KUKA KRL program: EPS_2_25694_AC01A_A_20260223033028.src

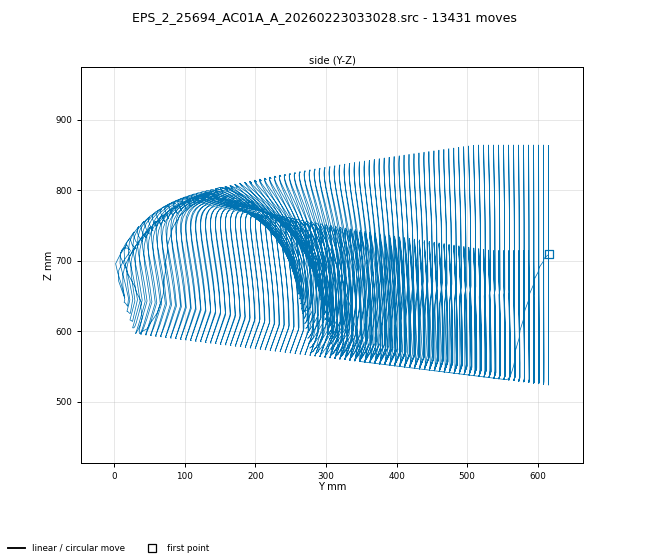
[picture p0: tool path of EPS_2_25694_AC01A_A_20260223033028.src, 13431 of 13433 moves have a stored position in this frame; points joined in program order, loops and branches not executed]
&ACCESS RVP
&REL 4
&COMMENT QRS 19112012
&PARAM EDITMASK = *
DEF PART()
EXT BAS (BAS_COMMAND :IN,REAL :IN )
INT I
BAS (#INITMOV,0 )

;KUKA QRS Post kuka4.cps  Date:22-06-2017 !

File_ID=3047

QRS_PRE_INIT()

;Init var - Until changes are made in qrs_pre_init
Outlet_Square_prg=0
Inlet_1_Square_prg=0
Inlet_2_Square_prg=0
Inlet_3_Square_prg=0
Inlet_4_Square_prg=0
Inlet_5_Square_prg=0

Outlet_1={X 0.000, Y 513.730, Z 763.500, B 0.000, E1 0.000 }
Inlet_1={X 0.000, Y 535.920, Z 314.500, B 0.000, E1 93.000 }
Inlet_2={X 0.000, Y 525.250, Z 538.500, B 0.000, E1 257.000 }
Outlet_1_type=201
Inlet_1_type=299
Inlet_2_type=251
;QRS#1=Sidecore dimensions
;QRS#2=200-8" PVC SDR 35
;QRS#3=300-12" PVC SDR 35
;QRS#4=250-10" PVC SDR 35
;QRS#5=
;QRS#6=
;QRS#7=
;QRS#8=
;QRS#9=12-08 PSX
;QRS#10=16M PSX
;QRS#11=14M PSX
;QRS#12=
;QRS#13=
;QRS#14=
;QRS#15=
;QRS#16=1220x127x1143 3,75'
;QRS#17=EPS Height
;QRS#18=864
;QRS#19=*
;QRS#20= UPDATED VERSION 22-06-2017
;QRS#21=*
Outlet_Square=0100
Inlet_1_Square=0150
Inlet_2_Square=0100
Inlet_3_Square=0
Inlet_4_Square=0
Inlet_5_Square=0
Mill_Square=1
Outlet_Square_Prg=204
Inlet_1_Square_prg=206
Inlet_2_Square_prg=205

QRS_INIT()

$ADVANCE=5

; T1
PTP {E1 173.417,E2 173.417}
PTP {X 0,Y 615.495,A -85,B 0,C 180,E1 173.417,E2 173.417,E3 0,E4 0,E5 0,E6 0}
QRS_SPEED_INIT()
LIN {X 0,Y 615.495,Z 709.245,A -85,B 0,C 180,E1 173.417,E2 173.417,E3 0,E4 0,E5 0,E6 0} C_VEL
LIN {X 0,Y 615.493,Z 705.573,A -85,B 0,C 180,E1 172.125,E2 172.125} C_VEL
LIN {X 0,Y 615.497,Z 700.547,A -85,B 0,C 180,E1 170.802,E2 170.802} C_VEL
LIN {X 0,Y 615.496,Z 694.074,A -85,B 0,C 180,E1 169.474,E2 169.474} C_VEL
LIN {X 0,Y 615.496,Z 685.953,A -85,B 0,C 180,E1 168.14,E2 168.14} C_VEL
LIN {X 0,Y 615.496,Z 677.25,A -85,B 0,C 180,E1 166.967,E2 166.967} C_VEL
LIN {X 0,Y 615.496,Z 667.933,A -85,B 0,C 180,E1 165.912,E2 165.912} C_VEL
LIN {X 0,Y 615.497,Z 657.856,A -85,B 0,C 180,E1 164.944,E2 164.944} C_VEL
LIN {X 0,Y 615.499,Z 645.706,A -85,B 0,C 180,E1 163.964,E2 163.964} C_VEL
LIN {X 0,Y 615.497,Z 633.795,A -85,B 0,C 180,E1 163.158,E2 163.158} C_VEL
LIN {X 0,Y 615.489,Z 621.694,A -85,B 0,C 180,E1 162.473,E2 162.473} C_VEL
LIN {X 0,Y 615.478,Z 607.053,A -85,B 0,C 180,E1 161.801,E2 161.801} C_VEL
LIN {X 0,Y 615.487,Z 591.984,A -85,B 0,C 180,E1 161.268,E2 161.268} C_VEL
LIN {X 0,Y 615.48,Z 576.911,A -85,B 0,C 180,E1 160.879,E2 160.879} C_VEL
LIN {X 0,Y 615.476,Z 561.369,A -85,B 0,C 180,E1 160.619,E2 160.619} C_VEL
LIN {X 0,Y 615.5,Z 523.699,A -85,B 0,C 180,E1 160.164,E2 160.164} C_VEL
LIN {X 0,Y 615.486,Z 523.681,A -85,B 0,C 180,E1 157.156,E2 157.156} C_VEL
LIN {X 0,Y 615.484,Z 523.694,A -85,B 0,C 180,E1 154.284,E2 154.284} C_VEL
LIN {X 0,Y 615.478,Z 523.69,A -85,B 0,C 180,E1 151.552,E2 151.552} C_VEL
LIN {X 0,Y 615.484,Z 523.682,A -85,B 0,C 180,E1 148.915,E2 148.915} C_VEL
LIN {X 0,Y 615.496,Z 523.697,A -85,B 0,C 180,E1 145.979,E2 145.979} C_VEL
LIN {X 0,Y 615.487,Z 523.682,A -85,B 0,C 180,E1 143.064,E2 143.064} C_VEL
LIN {X 0,Y 615.477,Z 523.69,A -85,B 0,C 180,E1 140.249,E2 140.249} C_VEL
LIN {X 0,Y 615.493,Z 523.698,A -85,B 0,C 180,E1 137.648,E2 137.648} C_VEL
LIN {X 0,Y 615.481,Z 523.684,A -85,B 0,C 180,E1 134.931,E2 134.931} C_VEL
LIN {X 0,Y 615.477,Z 523.69,A -85,B 0,C 180,E1 132.08,E2 132.08} C_VEL
LIN {X 0,Y 615.492,Z 523.695,A -85,B 0,C 180,E1 129.75,E2 129.75} C_VEL
LIN {X 0,Y 615.482,Z 523.686,A -85,B 0,C 180,E1 126.936,E2 126.936} C_VEL
LIN {X 0,Y 615.49,Z 523.681,A -85,B 0,C 180,E1 124.702,E2 124.702} C_VEL
LIN {X 0,Y 615.484,Z 523.682,A -85,B 0,C 180,E1 122.331,E2 122.331} C_VEL
LIN {X 0,Y 615.495,Z 523.701,A -85,B 0,C 180,E1 119.406,E2 119.406} C_VEL
LIN {X 0,Y 615.492,Z 523.68,A -85,B 0,C 180,E1 116.444,E2 116.444} C_VEL
LIN {X 0,Y 615.487,Z 523.693,A -85,B 0,C 180,E1 113.557,E2 113.557} C_VEL
LIN {X 0,Y 615.481,Z 523.688,A -85,B 0,C 180,E1 110.731,E2 110.731} C_VEL
LIN {X 0,Y 615.478,Z 523.684,A -85,B 0,C 180,E1 107.958,E2 107.958} C_VEL
LIN {X 0,Y 615.495,Z 523.698,A -85,B 0,C 180,E1 105.226,E2 105.226} C_VEL
LIN {X 0,Y 615.483,Z 523.686,A -85,B 0,C 180,E1 102.531,E2 102.531} C_VEL
LIN {X 0,Y 615.48,Z 523.683,A -85,B 0,C 180,E1 99.863,E2 99.863} C_VEL
LIN {X 0,Y 615.49,Z 523.694,A -85,B 0,C 180,E1 97.216,E2 97.216} C_VEL
LIN {X 0,Y 615.481,Z 523.692,A -85,B 0,C 180,E1 94.585,E2 94.585} C_VEL
LIN {X 0,Y 615.494,Z 523.68,A -85,B 0,C 180,E1 91.963,E2 91.963} C_VEL
LIN {X 0,Y 615.476,Z 523.689,A -85,B 0,C 180,E1 89.346,E2 89.346} C_VEL
LIN {X 0,Y 615.492,Z 523.699,A -85,B 0,C 180,E1 86.727,E2 86.727} C_VEL
LIN {X 0,Y 615.487,Z 523.684,A -85,B 0,C 180,E1 84.102,E2 84.102} C_VEL
LIN {X 0,Y 615.477,Z 523.685,A -85,B 0,C 180,E1 81.464,E2 81.464} C_VEL
LIN {X 0,Y 615.498,Z 523.694,A -85,B 0,C 180,E1 78.808,E2 78.808} C_VEL
LIN {X 0,Y 615.485,Z 523.686,A -85,B 0,C 180,E1 76.067,E2 76.067} C_VEL
LIN {X 0,Y 615.478,Z 523.684,A -85,B 0,C 180,E1 73.414,E2 73.414} C_VEL
LIN {X 0,Y 615.492,Z 523.696,A -85,B 0,C 180,E1 70.663,E2 70.663} C_VEL
LIN {X 0,Y 615.491,Z 523.681,A -85,B 0,C 180,E1 67.652,E2 67.652} C_VEL
LIN {X 0,Y 615.475,Z 523.687,A -85,B 0,C 180,E1 65.008,E2 65.008} C_VEL
LIN {X 0,Y 615.481,Z 523.689,A -85,B 0,C 180,E1 62.823,E2 62.823} C_VEL
LIN {X 0,Y 615.492,Z 523.698,A -85,B 0,C 180,E1 60.204,E2 60.204} C_VEL
LIN {X 0,Y 615.491,Z 523.682,A -85,B 0,C 180,E1 57.543,E2 57.543} C_VEL
LIN {X 0,Y 615.482,Z 523.682,A -85,B 0,C 180,E1 55.185,E2 55.185} C_VEL
LIN {X 0,Y 615.475,Z 523.688,A -85,B 0,C 180,E1 52.758,E2 52.758} C_VEL
LIN {X 0,Y 615.488,Z 523.695,A -85,B 0,C 180,E1 49.91,E2 49.91} C_VEL
LIN {X 0,Y 615.485,Z 523.689,A -85,B 0,C 180,E1 47.647,E2 47.647} C_VEL
LIN {X 0,Y 615.478,Z 523.683,A -85,B 0,C 180,E1 44.931,E2 44.931} C_VEL
LIN {X 0,Y 615.498,Z 523.696,A -85,B 0,C 180,E1 42.082,E2 42.082} C_VEL
LIN {X 0,Y 615.492,Z 523.68,A -85,B 0,C 180,E1 39.063,E2 39.063} C_VEL
LIN {X 0,Y 615.479,Z 523.687,A -85,B 0,C 180,E1 36.425,E2 36.425} C_VEL
LIN {X 0,Y 615.487,Z 523.692,A -85,B 0,C 180,E1 33.535,E2 33.535} C_VEL
LIN {X 0,Y 615.485,Z 523.682,A -85,B 0,C 180,E1 30.919,E2 30.919} C_VEL
LIN {X 0,Y 615.476,Z 523.685,A -85,B 0,C 180,E1 28.449,E2 28.449} C_VEL
LIN {X 0,Y 615.496,Z 523.701,A -85,B 0,C 180,E1 27.706,E2 27.706} C_VEL
LIN {X 0,Y 615.489,Z 531.805,A -85,B 0,C 180,E1 27.591,E2 27.591} C_VEL
LIN {X 0,Y 615.495,Z 589.214,A -85,B 0,C 180,E1 26.895,E2 26.895} C_VEL
LIN {X 0,Y 615.478,Z 603.233,A -85,B 0,C 180,E1 26.595,E2 26.595} C_VEL
LIN {X 0,Y 615.483,Z 616.816,A -85,B 0,C 180,E1 26.17,E2 26.17} C_VEL
LIN {X 0,Y 615.496,Z 629.536,A -85,B 0,C 180,E1 25.643,E2 25.643} C_VEL
LIN {X 0,Y 615.491,Z 641.959,A -85,B 0,C 180,E1 24.991,E2 24.991} C_VEL
LIN {X 0,Y 615.498,Z 653.128,A -85,B 0,C 180,E1 24.271,E2 24.271} C_VEL
LIN {X 0,Y 615.499,Z 664.53,A -85,B 0,C 180,E1 23.377,E2 23.377} C_VEL
LIN {X 0,Y 615.492,Z 675.308,A -85,B 0,C 180,E1 22.348,E2 22.348} C_VEL
LIN {X 0,Y 615.496,Z 684.638,A -85,B 0,C 180,E1 21.256,E2 21.256} C_VEL
LIN {X 0,Y 615.494,Z 691.433,A -85,B 0,C 180,E1 20.296,E2 20.296} C_VEL
LIN {X 0,Y 615.495,Z 697.081,A -85,B 0,C 180,E1 19.337,E2 19.337} C_VEL
LIN {X 0,Y 615.495,Z 702.21,A -85,B 0,C 180,E1 18.282,E2 18.282} C_VEL
LIN {X 0,Y 615.496,Z 707.259,A -85,B 0,C 180,E1 16.928,E2 16.928} C_VEL
LIN {X 0,Y 615.494,Z 710.032,A -85,B 0,C 180,E1 15.905,E2 15.905} C_VEL
LIN {X 0,Y 615.496,Z 712.389,A -85,B 0,C 180,E1 14.549,E2 14.549} C_VEL
LIN {X 0,Y 615.489,Z 713.337,A -85,B 0,C 180,E1 13.201,E2 13.201} C_VEL
LIN {X 0,Y 615.495,Z 712.911,A -85,B 0,C 180,E1 11.86,E2 11.86} C_VEL
LIN {X 0,Y 615.496,Z 711.131,A -85,B 0,C 180,E1 10.526,E2 10.526} C_VEL
LIN {X 0,Y 615.496,Z 707.948,A -85,B 0,C 180,E1 9.198,E2 9.198} C_VEL
LIN {X 0,Y 615.493,Z 703.274,A -85,B 0,C 180,E1 7.875,E2 7.875} C_VEL
LIN {X 0,Y 615.497,Z 696.991,A -85,B 0,C 180,E1 6.556,E2 6.556} C_VEL
LIN {X 0,Y 615.495,Z 690.024,A -85,B 0,C 180,E1 5.405,E2 5.405} C_VEL
LIN {X 0,Y 615.497,Z 681.428,A -85,B 0,C 180,E1 4.256,E2 4.256} C_VEL
LIN {X 0,Y 615.496,Z 672.486,A -85,B 0,C 180,E1 3.273,E2 3.273} C_VEL
LIN {X 0,Y 615.499,Z 661.696,A -85,B 0,C 180,E1 2.29,E2 2.29} C_VEL
LIN {X 0,Y 615.498,Z 650.756,A -85,B 0,C 180,E1 1.472,E2 1.472} C_VEL
LIN {X 0,Y 615.488,Z 638.756,A -85,B 0,C 180,E1 0.736,E2 0.736} C_VEL
LIN {X 0,Y 615.485,Z 625.402,A -85,B 0,C 180,E1 0.081,E2 0.081} C_VEL
LIN {X 0,Y 615.495,Z 611.227,A -85,B 0,C 180,E1 -0.45,E2 -0.45} C_VEL
LIN {X 0,Y 615.48,Z 597.695,A -85,B 0,C 180,E1 -0.818,E2 -0.818} C_VEL
LIN {X 0,Y 615.476,Z 583.862,A -85,B 0,C 180,E1 -1.064,E2 -1.064} C_VEL
LIN {X 0,Y 615.488,Z 523.701,A -85,B 0,C 180,E1 -1.779,E2 -1.779} C_VEL
LIN {X 0,Y 615.497,Z 523.68,A -85,B 0,C 180,E1 -4.585,E2 -4.585} C_VEL
LIN {X 0,Y 615.477,Z 523.691,A -85,B 0,C 180,E1 -7.216,E2 -7.216} C_VEL
LIN {X 0,Y 615.485,Z 523.695,A -85,B 0,C 180,E1 -9.863,E2 -9.863} C_VEL
LIN {X 0,Y 615.486,Z 523.683,A -85,B 0,C 180,E1 -12.53,E2 -12.53} C_VEL
LIN {X 0,Y 615.478,Z 523.694,A -85,B 0,C 180,E1 -15.227,E2 -15.227} C_VEL
LIN {X 0,Y 615.487,Z 523.689,A -85,B 0,C 180,E1 -17.957,E2 -17.957} C_VEL
LIN {X 0,Y 615.49,Z 523.683,A -85,B 0,C 180,E1 -20.731,E2 -20.731} C_VEL
LIN {X 0,Y 615.489,Z 523.699,A -85,B 0,C 180,E1 -23.557,E2 -23.557} C_VEL
LIN {X 0,Y 615.494,Z 523.691,A -85,B 0,C 180,E1 -25.716,E2 -25.716} C_VEL
LIN {X 0,Y 615.476,Z 523.685,A -85,B 0,C 180,E1 -28.449,E2 -28.449} C_VEL
LIN {X 0,Y 615.491,Z 523.692,A -85,B 0,C 180,E1 -31.088,E2 -31.088} C_VEL
LIN {X 0,Y 615.497,Z 523.682,A -85,B 0,C 180,E1 -34.022,E2 -34.022} C_VEL
LIN {X 0,Y 615.482,Z 523.692,A -85,B 0,C 180,E1 -36.937,E2 -36.937} C_VEL
LIN {X 0,Y 615.481,Z 523.689,A -85,B 0,C 180,E1 -39.751,E2 -39.751} C_VEL
LIN {X 0,Y 615.488,Z 523.682,A -85,B 0,C 180,E1 -42.353,E2 -42.353} C_VEL
LIN {X 0,Y 615.488,Z 523.698,A -85,B 0,C 180,E1 -45.069,E2 -45.069} C_VEL
LIN {X 0,Y 615.477,Z 523.686,A -85,B 0,C 180,E1 -47.921,E2 -47.921} C_VEL
LIN {X 0,Y 615.493,Z 523.681,A -85,B 0,C 180,E1 -50.251,E2 -50.251} C_VEL
LIN {X 0,Y 615.492,Z 523.701,A -85,B 0,C 180,E1 -53.063,E2 -53.063} C_VEL
LIN {X 0,Y 615.497,Z 523.692,A -85,B 0,C 180,E1 -55.299,E2 -55.299} C_VEL
LIN {X 0,Y 615.484,Z 523.686,A -85,B 0,C 180,E1 -57.67,E2 -57.67} C_VEL
LIN {X 0,Y 615.483,Z 523.872,A -85,B 0,C 180,E1 -60.304,E2 -60.304} C_VEL
LIN {X 0,Y 615.491,Z 544.028,A -85,B 0,C 180,E1 -63.106,E2 -63.106} C_VEL
LIN {X 0,Y 615.489,Z 563.357,A -85,B 0,C 180,E1 -65.729,E2 -65.729} C_VEL
LIN {X 0,Y 615.494,Z 584.743,A -85,B 0,C 180,E1 -68.569,E2 -68.569} C_VEL
LIN {X 0,Y 615.488,Z 606.431,A -85,B 0,C 180,E1 -71.396,E2 -71.396} C_VEL
LIN {X 0,Y 615.479,Z 627.455,A -85,B 0,C 180,E1 -74.095,E2 -74.095} C_VEL
LIN {X 0,Y 615.492,Z 650.105,A -85,B 0,C 180,E1 -76.967,E2 -76.967} C_VEL
LIN {X 0,Y 615.488,Z 651.269,A -85,B 0,C 180,E1 -77.114,E2 -77.114} C_VEL
LIN {X 0,Y 615.489,Z 759.854,A -85,B 0,C 180,E1 -78.411,E2 -78.411} C_VEL
LIN {X 0,Y 615.492,Z 772.359,A -85,B 0,C 180,E1 -78.682,E2 -78.682} C_VEL
LIN {X 0,Y 615.496,Z 785.512,A -85,B 0,C 180,E1 -79.109,E2 -79.109} C_VEL
LIN {X 0,Y 615.484,Z 797.486,A -85,B 0,C 180,E1 -79.64,E2 -79.64} C_VEL
LIN {X 0,Y 615.483,Z 809.002,A -85,B 0,C 180,E1 -80.304,E2 -80.304} C_VEL
LIN {X 0,Y 615.499,Z 819.346,A -85,B 0,C 180,E1 -81.05,E2 -81.05} C_VEL
LIN {X 0,Y 615.497,Z 827.816,A -85,B 0,C 180,E1 -81.795,E2 -81.795} C_VEL
LIN {X 0,Y 615.498,Z 835.61,A -85,B 0,C 180,E1 -82.62,E2 -82.62} C_VEL
LIN {X 0,Y 615.496,Z 843.206,A -85,B 0,C 180,E1 -83.608,E2 -83.608} C_VEL
LIN {X 0,Y 615.498,Z 850.207,A -85,B 0,C 180,E1 -84.759,E2 -84.759} C_VEL
LIN {X 0,Y 615.494,Z 854.853,A -85,B 0,C 180,E1 -85.744,E2 -85.744} C_VEL
LIN {X 0,Y 615.496,Z 858.4,A -85,B 0,C 180,E1 -86.727,E2 -86.727} C_VEL
LIN {X 0,Y 615.497,Z 860.234,A -85,B 0,C 180,E1 -87.383,E2 -87.383} C_VEL
LIN {X 0,Y 615.496,Z 861.609,A -85,B 0,C 180,E1 -88.037,E2 -88.037} C_VEL
LIN {X 0,Y 615.496,Z 863.174,A -85,B 0,C 180,E1 -89.346,E2 -89.346} C_VEL
LIN {X 0,Y 615.494,Z 863.389,A -85,B 0,C 180,E1 -90,E2 -90} C_VEL
LIN {X 0,Y 615.496,Z 862.579,A -85,B 0,C 180,E1 -91.309,E2 -91.309} C_VEL
LIN {X 0,Y 615.496,Z 861.608,A -85,B 0,C 180,E1 -91.963,E2 -91.963} C_VEL
LIN {X 0,Y 615.497,Z 860.232,A -85,B 0,C 180,E1 -92.618,E2 -92.618} C_VEL
LIN {X 0,Y 615.496,Z 857.348,A -85,B 0,C 180,E1 -93.601,E2 -93.601} C_VEL
LIN {X 0,Y 615.498,Z 853.44,A -85,B 0,C 180,E1 -94.585,E2 -94.585} C_VEL
LIN {X 0,Y 615.499,Z 848.403,A -85,B 0,C 180,E1 -95.57,E2 -95.57} C_VEL
LIN {X 0,Y 615.497,Z 841.87,A -85,B 0,C 180,E1 -96.583,E2 -96.583} C_VEL
LIN {X 0,Y 615.497,Z 834.13,A -85,B 0,C 180,E1 -97.546,E2 -97.546} C_VEL
LIN {X 0,Y 615.498,Z 826.041,A -85,B 0,C 180,E1 -98.371,E2 -98.371} C_VEL
LIN {X 0,Y 615.499,Z 816.163,A -85,B 0,C 180,E1 -99.199,E2 -99.199} C_VEL
LIN {X 0,Y 615.486,Z 804.975,A -85,B 0,C 180,E1 -99.946,E2 -99.946} C_VEL
LIN {X 0,Y 615.483,Z 794.015,A -85,B 0,C 180,E1 -100.527,E2 -100.527} C_VEL
LIN {X 0,Y 615.496,Z 781.426,A -85,B 0,C 180,E1 -101.042,E2 -101.042} C_VEL
LIN {X 0,Y 615.49,Z 769.049,A -85,B 0,C 180,E1 -101.402,E2 -101.402} C_VEL
LIN {X 0,Y 615.49,Z 755.439,A -85,B 0,C 180,E1 -101.652,E2 -101.652} C_VEL
LIN {X 0,Y 615.488,Z 651.263,A -85,B 0,C 180,E1 -102.887,E2 -102.887} C_VEL
LIN {X 0,Y 615.482,Z 630.116,A -85,B 0,C 180,E1 -105.566,E2 -105.566} C_VEL
LIN {X 0,Y 615.498,Z 608.936,A -85,B 0,C 180,E1 -108.28,E2 -108.28} C_VEL
LIN {X 0,Y 615.497,Z 587.409,A -85,B 0,C 180,E1 -111.081,E2 -111.081} C_VEL
LIN {X 0,Y 615.476,Z 567.021,A -85,B 0,C 180,E1 -113.781,E2 -113.781} C_VEL
LIN {X 0,Y 615.496,Z 546.216,A -85,B 0,C 180,E1 -116.594,E2 -116.594} C_VEL
LIN {X 0,Y 615.497,Z 525.925,A -85,B 0,C 180,E1 -119.406,E2 -119.406} C_VEL
LIN {X 0,Y 615.479,Z 523.686,A -85,B 0,C 180,E1 -119.744,E2 -119.744} C_VEL
LIN {X 0,Y 615.487,Z 523.688,A -85,B 0,C 180,E1 -122.458,E2 -122.458} C_VEL
LIN {X 0,Y 615.497,Z 523.696,A -85,B 0,C 180,E1 -124.815,E2 -124.815} C_VEL
LIN {X 0,Y 615.486,Z 523.691,A -85,B 0,C 180,E1 -127.243,E2 -127.243} C_VEL
LIN {X 0,Y 615.477,Z 523.686,A -85,B 0,C 180,E1 -130.087,E2 -130.087} C_VEL
LIN {X 0,Y 615.478,Z 523.691,A -85,B 0,C 180,E1 -132.354,E2 -132.354} C_VEL
LIN {X 0,Y 615.481,Z 523.694,A -85,B 0,C 180,E1 -135.069,E2 -135.069} C_VEL
LIN {X 0,Y 615.491,Z 523.682,A -85,B 0,C 180,E1 -137.92,E2 -137.92} C_VEL
LIN {X 0,Y 615.492,Z 523.693,A -85,B 0,C 180,E1 -140.938,E2 -140.938} C_VEL
LIN {X 0,Y 615.478,Z 523.685,A -85,B 0,C 180,E1 -143.574,E2 -143.574} C_VEL
LIN {X 0,Y 615.489,Z 523.697,A -85,B 0,C 180,E1 -146.466,E2 -146.466} C_VEL
LIN {X 0,Y 615.487,Z 523.687,A -85,B 0,C 180,E1 -149.08,E2 -149.08} C_VEL
LIN {X 0,Y 615.476,Z 523.685,A -85,B 0,C 180,E1 -151.552,E2 -151.552} C_VEL
LIN {X 0,Y 615.498,Z 523.699,A -85,B 0,C 180,E1 -154.43,E2 -154.43} C_VEL
LIN {X 0,Y 615.486,Z 523.684,A -85,B 0,C 180,E1 -157.155,E2 -157.155} C_VEL
LIN {X 0,Y 615.485,Z 523.69,A -85,B 0,C 180,E1 -159.967,E2 -159.967} C_VEL
LIN {X 0,Y 615.48,Z 523.692,A -85,B 0,C 180,E1 -162.729,E2 -162.729} C_VEL
LIN {X 0,Y 615.48,Z 523.684,A -85,B 0,C 180,E1 -165.45,E2 -165.45} C_VEL
LIN {X 0,Y 615.487,Z 523.701,A -85,B 0,C 180,E1 -166.252,E2 -166.252} C_VEL
LIN {X 0,Y 615.476,Z 569.038,A -85,B 0,C 180,E1 -166.819,E2 -166.819} C_VEL
LIN {X 0,Y 615.485,Z 583.996,A -85,B 0,C 180,E1 -167.134,E2 -167.134} C_VEL
LIN {X 0,Y 615.479,Z 599.217,A -85,B 0,C 180,E1 -167.595,E2 -167.595} C_VEL
LIN {X 0,Y 615.486,Z 612.817,A -85,B 0,C 180,E1 -168.139,E2 -168.139} C_VEL
LIN {X 0,Y 615.493,Z 626.215,A -85,B 0,C 180,E1 -168.807,E2 -168.807} C_VEL
LIN {X 0,Y 615.5,Z 638.582,A -85,B 0,C 180,E1 -169.556,E2 -169.556} C_VEL
LIN {X 0,Y 615.499,Z 651.123,A -85,B 0,C 180,E1 -170.47,E2 -170.47} C_VEL
LIN {X 0,Y 615.496,Z 662.521,A -85,B 0,C 180,E1 -171.463,E2 -171.463} C_VEL
LIN {X 0,Y 615.495,Z 672.115,A -85,B 0,C 180,E1 -172.454,E2 -172.454} C_VEL
LIN {X 0,Y 615.494,Z 681.536,A -85,B 0,C 180,E1 -173.608,E2 -173.608} C_VEL
LIN {X 0,Y 615.494,Z 690.39,A -85,B 0,C 180,E1 -174.923,E2 -174.923} C_VEL
LIN {X 0,Y 615.492,Z 696.739,A -85,B 0,C 180,E1 -176.071,E2 -176.071} C_VEL
LIN {X 0,Y 615.496,Z 702.589,A -85,B 0,C 180,E1 -177.382,E2 -177.382} C_VEL
LIN {X 0,Y 615.496,Z 707.094,A -85,B 0,C 180,E1 -178.691,E2 -178.691} C_VEL
LIN {X 0,Y 615.49,Z 710.314,A -85,B 0,C 180,E1 -180,E2 -180} C_VEL
LIN {X 0,Y 615.491,Z 712.362,A -85,B 0,C 180,E1 -181.308,E2 -181.308} C_VEL
LIN {X 0,Y 615.497,Z 713.291,A -85,B 0,C 180,E1 -182.618,E2 -182.618} C_VEL
LIN {X 0,Y 615.488,Z 713.108,A -85,B 0,C 180,E1 -183.928,E2 -183.928} C_VEL
LIN {X 0,Y 615.489,Z 711.806,A -85,B 0,C 180,E1 -185.241,E2 -185.241} C_VEL
LIN {X 0,Y 615.495,Z 709.245,A -85,B 0,C 180,E1 -186.583,E2 -186.583} C_VEL
LIN {X 0,Y 614.809,Z 708.026,A -85,B 0,C 180,E1 -187.114,E2 -187.114} C_VEL
LIN {X 0,Y 611.951,Z 705.822,A -85,B 0,C 180,E1 -187.974,E2 -187.974} C_VEL
LIN {X 0,Y 609.544,Z 703.512,A -85,B 0,C 180,E1 -188.657,E2 -188.657} C_VEL
LIN {X 0,Y 608.513,Z 701.422,A -85,B 0,C 180,E1 -189.174,E2 -189.174} C_VEL
LIN {X 0,Y 608.428,Z 700.673,A -85,B 0,C 180,E1 -189.347,E2 -189.347} C_VEL
LIN {X 0,Y 608.436,Z 694.266,A -85,B 0,C 180,E1 -190.65,E2 -190.65} C_VEL
LIN {X 0,Y 608.462,Z 687.154,A -85,B 0,C 180,E1 -191.83,E2 -191.83} C_VEL
LIN {X 0,Y 608.465,Z 678.57,A -85,B 0,C 180,E1 -193.016,E2 -193.016} C_VEL
LIN {X 0,Y 608.485,Z 668.197,A -85,B 0,C 180,E1 -194.207,E2 -194.207} C_VEL
LIN {X 0,Y 608.495,Z 657.544,A -85,B 0,C 180,E1 -195.233,E2 -195.233} C_VEL
LIN {X 0,Y 608.537,Z 645.262,A -85,B 0,C 180,E1 -196.225,E2 -196.225} C_VEL
LIN {X 0,Y 608.555,Z 631.774,A -85,B 0,C 180,E1 -197.127,E2 -197.127} C_VEL
LIN {X 0,Y 608.578,Z 617.426,A -85,B 0,C 180,E1 -197.907,E2 -197.907} C_VEL
LIN {X 0,Y 608.615,Z 603.979,A -85,B 0,C 180,E1 -198.493,E2 -198.493} C_VEL
LIN {X 0,Y 608.657,Z 589.173,A -85,B 0,C 180,E1 -198.994,E2 -198.994} C_VEL
LIN {X 0,Y 608.663,Z 573.906,A -85,B 0,C 180,E1 -199.366,E2 -199.366} C_VEL
LIN {X 0,Y 608.67,Z 556.486,A -85,B 0,C 180,E1 -199.629,E2 -199.629} C_VEL
LIN {X 0,Y 608.53,Z 525.02,A -85,B 0,C 180,E1 -200.013,E2 -200.013} C_VEL
LIN {X 0,Y 608.469,Z 524.693,A -85,B 0,C 180,E1 -200.053,E2 -200.053} C_VEL
LIN {X 0,Y 608.461,Z 524.688,A -85,B 0,C 180,E1 -202.476,E2 -202.476} C_VEL
LIN {X 0,Y 608.452,Z 524.688,A -85,B 0,C 180,E1 -204.571,E2 -204.571} C_VEL
LIN {X 0,Y 608.476,Z 524.684,A -85,B 0,C 180,E1 -207.206,E2 -207.206} C_VEL
LIN {X 0,Y 608.468,Z 524.695,A -85,B 0,C 180,E1 -209.971,E2 -209.971} C_VEL
LIN {X 0,Y 608.453,Z 524.687,A -85,B 0,C 180,E1 -212.879,E2 -212.879} C_VEL
LIN {X 0,Y 608.434,Z 524.689,A -85,B 0,C 180,E1 -215.278,E2 -215.278} C_VEL
LIN {X 0,Y 608.472,Z 524.688,A -85,B 0,C 180,E1 -217.746,E2 -217.746} C_VEL
LIN {X 0,Y 608.453,Z 524.696,A -85,B 0,C 180,E1 -220.329,E2 -220.329} C_VEL
LIN {X 0,Y 608.484,Z 524.683,A -85,B 0,C 180,E1 -223.31,E2 -223.31} C_VEL
LIN {X 0,Y 608.465,Z 524.693,A -85,B 0,C 180,E1 -226.13,E2 -226.13} C_VEL
LIN {X 0,Y 608.451,Z 524.691,A -85,B 0,C 180,E1 -228.823,E2 -228.823} C_VEL
LIN {X 0,Y 608.464,Z 524.685,A -85,B 0,C 180,E1 -231.411,E2 -231.411} C_VEL
LIN {X 0,Y 608.445,Z 524.69,A -85,B 0,C 180,E1 -233.954,E2 -233.954} C_VEL
LIN {X 0,Y 608.467,Z 524.692,A -85,B 0,C 180,E1 -236.329,E2 -236.329} C_VEL
LIN {X 0,Y 608.46,Z 524.694,A -85,B 0,C 180,E1 -238.73,E2 -238.73} C_VEL
LIN {X 0,Y 608.474,Z 524.685,A -85,B 0,C 180,E1 -241.379,E2 -241.379} C_VEL
LIN {X 0,Y 608.443,Z 524.689,A -85,B 0,C 180,E1 -243.964,E2 -243.964} C_VEL
LIN {X 0,Y 608.461,Z 524.688,A -85,B 0,C 180,E1 -246.155,E2 -246.155} C_VEL
LIN {X 0,Y 608.471,Z 524.688,A -85,B 0,C 180,E1 -248.308,E2 -248.308} C_VEL
LIN {X 0,Y 608.467,Z 524.688,A -85,B 0,C 180,E1 -251.284,E2 -251.284} C_VEL
LIN {X 0,Y 608.456,Z 524.686,A -85,B 0,C 180,E1 -253.906,E2 -253.906} C_VEL
LIN {X 0,Y 608.47,Z 524.691,A -85,B 0,C 180,E1 -256.643,E2 -256.643} C_VEL
LIN {X 0,Y 608.461,Z 524.69,A -85,B 0,C 180,E1 -259.35,E2 -259.35} C_VEL
LIN {X 0,Y 608.474,Z 524.684,A -85,B 0,C 180,E1 -262.033,E2 -262.033} C_VEL
LIN {X 0,Y 608.465,Z 524.69,A -85,B 0,C 180,E1 -264.698,E2 -264.698} C_VEL
LIN {X 0,Y 608.475,Z 524.69,A -85,B 0,C 180,E1 -267.352,E2 -267.352} C_VEL
LIN {X 0,Y 608.477,Z 524.684,A -85,B 0,C 180,E1 -270,E2 -270} C_VEL
LIN {X 0,Y 608.469,Z 524.687,A -85,B 0,C 180,E1 -272.648,E2 -272.648} C_VEL
LIN {X 0,Y 608.473,Z 524.695,A -85,B 0,C 180,E1 -275.301,E2 -275.301} C_VEL
LIN {X 0,Y 608.476,Z 524.685,A -85,B 0,C 180,E1 -277.967,E2 -277.967} C_VEL
LIN {X 0,Y 608.456,Z 524.687,A -85,B 0,C 180,E1 -280.65,E2 -280.65} C_VEL
LIN {X 0,Y 608.471,Z 524.695,A -85,B 0,C 180,E1 -283.356,E2 -283.356} C_VEL
LIN {X 0,Y 608.458,Z 524.687,A -85,B 0,C 180,E1 -286.093,E2 -286.093} C_VEL
LIN {X 0,Y 608.452,Z 524.688,A -85,B 0,C 180,E1 -288.869,E2 -288.869} C_VEL
LIN {X 0,Y 608.474,Z 524.693,A -85,B 0,C 180,E1 -291.691,E2 -291.691} C_VEL
LIN {X 0,Y 608.451,Z 524.687,A -85,B 0,C 180,E1 -294.571,E2 -294.571} C_VEL
LIN {X 0,Y 608.474,Z 524.688,A -85,B 0,C 180,E1 -297.207,E2 -297.207} C_VEL
LIN {X 0,Y 608.47,Z 524.691,A -85,B 0,C 180,E1 -299.973,E2 -299.973} C_VEL
LIN {X 0,Y 608.464,Z 524.686,A -85,B 0,C 180,E1 -302.523,E2 -302.523} C_VEL
LIN {X 0,Y 608.448,Z 524.69,A -85,B 0,C 180,E1 -305.277,E2 -305.277} C_VEL
LIN {X 0,Y 608.465,Z 524.689,A -85,B 0,C 180,E1 -308.241,E2 -308.241} C_VEL
LIN {X 0,Y 608.477,Z 524.687,A -85,B 0,C 180,E1 -310.332,E2 -310.332} C_VEL
LIN {X 0,Y 608.463,Z 524.687,A -85,B 0,C 180,E1 -313.309,E2 -313.309} C_VEL
LIN {X 0,Y 608.475,Z 524.693,A -85,B 0,C 180,E1 -316.132,E2 -316.132} C_VEL
LIN {X 0,Y 608.455,Z 524.687,A -85,B 0,C 180,E1 -318.824,E2 -318.824} C_VEL
LIN {X 0,Y 608.468,Z 524.686,A -85,B 0,C 180,E1 -321.412,E2 -321.412} C_VEL
LIN {X 0,Y 608.475,Z 524.692,A -85,B 0,C 180,E1 -323.95,E2 -323.95} C_VEL
LIN {X 0,Y 608.467,Z 524.693,A -85,B 0,C 180,E1 -326.33,E2 -326.33} C_VEL
LIN {X 0,Y 608.474,Z 524.687,A -85,B 0,C 180,E1 -328.727,E2 -328.727} C_VEL
LIN {X 0,Y 608.465,Z 524.685,A -85,B 0,C 180,E1 -331.38,E2 -331.38} C_VEL
LIN {X 0,Y 608.466,Z 524.694,A -85,B 0,C 180,E1 -332.145,E2 -332.145} C_VEL
LIN {X 0,Y 608.622,Z 556.104,A -85,B 0,C 180,E1 -332.53,E2 -332.53} C_VEL
LIN {X 0,Y 608.627,Z 589.449,A -85,B 0,C 180,E1 -332.948,E2 -332.948} C_VEL
LIN {X 0,Y 608.578,Z 603.495,A -85,B 0,C 180,E1 -333.255,E2 -333.255} C_VEL
LIN {X 0,Y 608.564,Z 616.069,A -85,B 0,C 180,E1 -333.648,E2 -333.648} C_VEL
LIN {X 0,Y 608.551,Z 629.667,A -85,B 0,C 180,E1 -334.214,E2 -334.214} C_VEL
LIN {X 0,Y 608.538,Z 642.325,A -85,B 0,C 180,E1 -334.886,E2 -334.886} C_VEL
LIN {X 0,Y 608.502,Z 654.708,A -85,B 0,C 180,E1 -335.703,E2 -335.703} C_VEL
LIN {X 0,Y 608.484,Z 665.932,A -85,B 0,C 180,E1 -336.608,E2 -336.608} C_VEL
LIN {X 0,Y 608.471,Z 676.055,A -85,B 0,C 180,E1 -337.595,E2 -337.595} C_VEL
LIN {X 0,Y 608.46,Z 685.081,A -85,B 0,C 180,E1 -338.664,E2 -338.664} C_VEL
LIN {X 0,Y 608.441,Z 692.491,A -85,B 0,C 180,E1 -339.725,E2 -339.725} C_VEL
LIN {X 0,Y 608.437,Z 698.556,A -85,B 0,C 180,E1 -340.78,E2 -340.78} C_VEL
LIN {X 0,Y 608.428,Z 703.431,A -85,B 0,C 180,E1 -341.828,E2 -341.828} C_VEL
LIN {X 0,Y 608.424,Z 707.298,A -85,B 0,C 180,E1 -342.87,E2 -342.87} C_VEL
LIN {X 0,Y 608.43,Z 710.263,A -85,B 0,C 180,E1 -343.906,E2 -343.906} C_VEL
LIN {X 0,Y 608.42,Z 712.809,A -85,B 0,C 180,E1 -345.278,E2 -345.278} C_VEL
LIN {X 0,Y 608.433,Z 713.912,A -85,B 0,C 180,E1 -346.643,E2 -346.643} C_VEL
LIN {X 0,Y 608.439,Z 713.626,A -85,B 0,C 180,E1 -348,E2 -348} C_VEL
LIN {X 0,Y 608.436,Z 711.969,A -85,B 0,C 180,E1 -349.35,E2 -349.35} C_VEL
LIN {X 0,Y 608.421,Z 708.912,A -85,B 0,C 180,E1 -350.694,E2 -350.694} C_VEL
LIN {X 0,Y 608.428,Z 704.394,A -85,B 0,C 180,E1 -352.033,E2 -352.033} C_VEL
LIN {X 0,Y 608.438,Z 699.92,A -85,B 0,C 180,E1 -353.034,E2 -353.034} C_VEL
LIN {X 0,Y 608.457,Z 693.492,A -85,B 0,C 180,E1 -354.2,E2 -354.2} C_VEL
LIN {X 0,Y 608.465,Z 685.548,A -85,B 0,C 180,E1 -355.363,E2 -355.363} C_VEL
LIN {X 0,Y 608.478,Z 677.282,A -85,B 0,C 180,E1 -356.358,E2 -356.358} C_VEL
LIN {X 0,Y 608.489,Z 667.392,A -85,B 0,C 180,E1 -357.352,E2 -357.352} C_VEL
LIN {X 0,Y 608.497,Z 656.422,A -85,B 0,C 180,E1 -358.263,E2 -358.263} C_VEL
LIN {X 0,Y 608.534,Z 644.213,A -85,B 0,C 180,E1 -359.09,E2 -359.09} C_VEL
LIN {X 0,Y 608.547,Z 632.216,A -85,B 0,C 180,E1 -359.752,E2 -359.752} C_VEL
LIN {X 0,Y 608.571,Z 619.003,A -85,B 0,C 180,E1 -360.331,E2 -360.331} C_VEL
LIN {X 0,Y 608.592,Z 604.509,A -85,B 0,C 180,E1 -360.807,E2 -360.807} C_VEL
LIN {X 0,Y 608.597,Z 590.813,A -85,B 0,C 180,E1 -361.117,E2 -361.117} C_VEL
LIN {X 0,Y 608.617,Z 565.495,A -85,B 0,C 180,E1 -361.448,E2 -361.448} C_VEL
LIN {X 0,Y 608.503,Z 525.017,A -85,B 0,C 180,E1 -361.934,E2 -361.934} C_VEL
LIN {X 0,Y 608.452,Z 524.695,A -85,B 0,C 180,E1 -361.945,E2 -361.945} C_VEL
LIN {X 0,Y 608.465,Z 524.686,A -85,B 0,C 180,E1 -364.638,E2 -364.638} C_VEL
LIN {X 0,Y 608.457,Z 524.691,A -85,B 0,C 180,E1 -367.3,E2 -367.3} C_VEL
LIN {X 0,Y 608.455,Z 524.692,A -85,B 0,C 180,E1 -369.978,E2 -369.978} C_VEL
LIN {X 0,Y 608.473,Z 524.685,A -85,B 0,C 180,E1 -372.677,E2 -372.677} C_VEL
LIN {X 0,Y 608.465,Z 524.694,A -85,B 0,C 180,E1 -375.406,E2 -375.406} C_VEL
LIN {X 0,Y 608.449,Z 524.689,A -85,B 0,C 180,E1 -378.172,E2 -378.172} C_VEL
LIN {X 0,Y 608.46,Z 524.689,A -85,B 0,C 180,E1 -380.982,E2 -380.982} C_VEL
LIN {X 0,Y 608.468,Z 524.69,A -85,B 0,C 180,E1 -383.845,E2 -383.845} C_VEL
LIN {X 0,Y 608.446,Z 524.69,A -85,B 0,C 180,E1 -386.036,E2 -386.036} C_VEL
LIN {X 0,Y 608.466,Z 524.686,A -85,B 0,C 180,E1 -388.62,E2 -388.62} C_VEL
LIN {X 0,Y 608.477,Z 524.694,A -85,B 0,C 180,E1 -391.316,E2 -391.316} C_VEL
LIN {X 0,Y 608.478,Z 524.688,A -85,B 0,C 180,E1 -393.737,E2 -393.737} C_VEL
LIN {X 0,Y 608.457,Z 524.687,A -85,B 0,C 180,E1 -396.092,E2 -396.092} C_VEL
LIN {X 0,Y 608.469,Z 524.686,A -85,B 0,C 180,E1 -398.588,E2 -398.588} C_VEL
LIN {X 0,Y 608.46,Z 524.695,A -85,B 0,C 180,E1 -401.343,E2 -401.343} C_VEL
LIN {X 0,Y 608.46,Z 524.686,A -85,B 0,C 180,E1 -404.265,E2 -404.265} C_VEL
LIN {X 0,Y 608.45,Z 524.696,A -85,B 0,C 180,E1 -407.041,E2 -407.041} C_VEL
LIN {X 0,Y 608.451,Z 524.69,A -85,B 0,C 180,E1 -409.697,E2 -409.697} C_VEL
LIN {X 0,Y 608.465,Z 524.686,A -85,B 0,C 180,E1 -412.254,E2 -412.254} C_VEL
LIN {X 0,Y 608.486,Z 524.694,A -85,B 0,C 180,E1 -415.09,E2 -415.09} C_VEL
LIN {X 0,Y 608.466,Z 524.686,A -85,B 0,C 180,E1 -417.906,E2 -417.906} C_VEL
LIN {X 0,Y 608.486,Z 524.818,A -85,B 0,C 180,E1 -420.063,E2 -420.063} C_VEL
LIN {X 0,Y 608.722,Z 528.605,A -85,B 0,C 180,E1 -420.615,E2 -420.615} C_VEL
LIN {X 0,Y 608.661,Z 548.654,A -85,B 0,C 180,E1 -423.421,E2 -423.421} C_VEL
LIN {X 0,Y 608.6,Z 568.704,A -85,B 0,C 180,E1 -426.161,E2 -426.161} C_VEL
LIN {X 0,Y 608.571,Z 588.753,A -85,B 0,C 180,E1 -428.846,E2 -428.846} C_VEL
LIN {X 0,Y 608.546,Z 610.22,A -85,B 0,C 180,E1 -431.668,E2 -431.668} C_VEL
LIN {X 0,Y 608.491,Z 631.525,A -85,B 0,C 180,E1 -434.423,E2 -434.423} C_VEL
LIN {X 0,Y 608.485,Z 651.491,A -85,B 0,C 180,E1 -436.974,E2 -436.974} C_VEL
LIN {X 0,Y 608.543,Z 759.97,A -85,B 0,C 180,E1 -438.277,E2 -438.277} C_VEL
LIN {X 0,Y 608.541,Z 773.231,A -85,B 0,C 180,E1 -438.572,E2 -438.572} C_VEL
LIN {X 0,Y 608.543,Z 786.344,A -85,B 0,C 180,E1 -439.01,E2 -439.01} C_VEL
LIN {X 0,Y 608.501,Z 797.643,A -85,B 0,C 180,E1 -439.52,E2 -439.52} C_VEL
LIN {X 0,Y 608.474,Z 809.203,A -85,B 0,C 180,E1 -440.191,E2 -440.191} C_VEL
LIN {X 0,Y 608.485,Z 819.599,A -85,B 0,C 180,E1 -440.946,E2 -440.946} C_VEL
LIN {X 0,Y 608.475,Z 828.116,A -85,B 0,C 180,E1 -441.699,E2 -441.699} C_VEL
LIN {X 0,Y 608.471,Z 835.964,A -85,B 0,C 180,E1 -442.534,E2 -442.534} C_VEL
LIN {X 0,Y 608.46,Z 843.288,A -85,B 0,C 180,E1 -443.485,E2 -443.485} C_VEL
LIN {X 0,Y 608.45,Z 848.868,A -85,B 0,C 180,E1 -444.366,E2 -444.366} C_VEL
LIN {X 0,Y 608.432,Z 853.952,A -85,B 0,C 180,E1 -445.363,E2 -445.363} C_VEL
LIN {X 0,Y 608.449,Z 857.897,A -85,B 0,C 180,E1 -446.358,E2 -446.358} C_VEL
LIN {X 0,Y 608.425,Z 860.81,A -85,B 0,C 180,E1 -447.352,E2 -447.352} C_VEL
LIN {X 0,Y 608.441,Z 862.202,A -85,B 0,C 180,E1 -448.015,E2 -448.015} C_VEL
LIN {X 0,Y 608.438,Z 863.784,A -85,B 0,C 180,E1 -449.339,E2 -449.339} C_VEL
LIN {X 0,Y 608.434,Z 864,A -85,B 0,C 180,E1 -450,E2 -450} C_VEL
LIN {X 0,Y 608.448,Z 863.183,A -85,B 0,C 180,E1 -451.324,E2 -451.324} C_VEL
LIN {X 0,Y 608.441,Z 862.201,A -85,B 0,C 180,E1 -451.986,E2 -451.986} C_VEL
LIN {X 0,Y 608.425,Z 860.808,A -85,B 0,C 180,E1 -452.649,E2 -452.649} C_VEL
LIN {X 0,Y 608.449,Z 857.895,A -85,B 0,C 180,E1 -453.643,E2 -453.643} C_VEL
LIN {X 0,Y 608.432,Z 853.948,A -85,B 0,C 180,E1 -454.638,E2 -454.638} C_VEL
LIN {X 0,Y 608.437,Z 847.874,A -85,B 0,C 180,E1 -455.801,E2 -455.801} C_VEL
LIN {X 0,Y 608.462,Z 841.232,A -85,B 0,C 180,E1 -456.8,E2 -456.8} C_VEL
LIN {X 0,Y 608.456,Z 832.986,A -85,B 0,C 180,E1 -457.801,E2 -457.801} C_VEL
LIN {X 0,Y 608.472,Z 824.532,A -85,B 0,C 180,E1 -458.636,E2 -458.636} C_VEL
LIN {X 0,Y 608.471,Z 814.086,A -85,B 0,C 180,E1 -459.474,E2 -459.474} C_VEL
LIN {X 0,Y 608.487,Z 803.749,A -85,B 0,C 180,E1 -460.145,E2 -460.145} C_VEL
LIN {X 0,Y 608.521,Z 792.239,A -85,B 0,C 180,E1 -460.741,E2 -460.741} C_VEL
LIN {X 0,Y 608.539,Z 779.871,A -85,B 0,C 180,E1 -461.225,E2 -461.225} C_VEL
LIN {X 0,Y 608.545,Z 766.424,A -85,B 0,C 180,E1 -461.597,E2 -461.597} C_VEL
LIN {X 0,Y 608.549,Z 754.056,A -85,B 0,C 180,E1 -461.808,E2 -461.808} C_VEL
LIN {X 0,Y 608.474,Z 651.401,A -85,B 0,C 180,E1 -463.038,E2 -463.038} C_VEL
LIN {X 0,Y 608.491,Z 631.519,A -85,B 0,C 180,E1 -465.577,E2 -465.577} C_VEL
LIN {X 0,Y 608.547,Z 610.215,A -85,B 0,C 180,E1 -468.333,E2 -468.333} C_VEL
LIN {X 0,Y 608.572,Z 588.747,A -85,B 0,C 180,E1 -471.155,E2 -471.155} C_VEL
LIN {X 0,Y 608.6,Z 568.697,A -85,B 0,C 180,E1 -473.84,E2 -473.84} C_VEL
LIN {X 0,Y 608.661,Z 548.648,A -85,B 0,C 180,E1 -476.579,E2 -476.579} C_VEL
LIN {X 0,Y 608.723,Z 528.598,A -85,B 0,C 180,E1 -479.386,E2 -479.386} C_VEL
LIN {X 0,Y 608.468,Z 524.715,A -85,B 0,C 180,E1 -479.953,E2 -479.953} C_VEL
LIN {X 0,Y 608.463,Z 524.69,A -85,B 0,C 180,E1 -482.522,E2 -482.522} C_VEL
LIN {X 0,Y 608.454,Z 524.692,A -85,B 0,C 180,E1 -485.277,E2 -485.277} C_VEL
LIN {X 0,Y 608.465,Z 524.686,A -85,B 0,C 180,E1 -487.747,E2 -487.747} C_VEL
LIN {X 0,Y 608.447,Z 524.691,A -85,B 0,C 180,E1 -490.328,E2 -490.328} C_VEL
LIN {X 0,Y 608.469,Z 524.688,A -85,B 0,C 180,E1 -493.308,E2 -493.308} C_VEL
LIN {X 0,Y 608.47,Z 524.687,A -85,B 0,C 180,E1 -496.13,E2 -496.13} C_VEL
LIN {X 0,Y 608.456,Z 524.696,A -85,B 0,C 180,E1 -498.823,E2 -498.823} C_VEL
LIN {X 0,Y 608.469,Z 524.686,A -85,B 0,C 180,E1 -501.412,E2 -501.412} C_VEL
LIN {X 0,Y 608.449,Z 524.689,A -85,B 0,C 180,E1 -503.955,E2 -503.955} C_VEL
LIN {X 0,Y 608.469,Z 524.691,A -85,B 0,C 180,E1 -506.329,E2 -506.329} C_VEL
LIN {X 0,Y 608.482,Z 524.692,A -85,B 0,C 180,E1 -508.727,E2 -508.727} C_VEL
LIN {X 0,Y 608.467,Z 524.686,A -85,B 0,C 180,E1 -511.382,E2 -511.382} C_VEL
LIN {X 0,Y 608.447,Z 524.691,A -85,B 0,C 180,E1 -513.964,E2 -513.964} C_VEL
LIN {X 0,Y 608.466,Z 524.691,A -85,B 0,C 180,E1 -516.155,E2 -516.155} C_VEL
LIN {X 0,Y 608.457,Z 524.689,A -85,B 0,C 180,E1 -519.018,E2 -519.018} C_VEL
LIN {X 0,Y 608.449,Z 524.69,A -85,B 0,C 180,E1 -521.828,E2 -521.828} C_VEL
LIN {X 0,Y 608.465,Z 524.692,A -85,B 0,C 180,E1 -524.594,E2 -524.594} C_VEL
LIN {X 0,Y 608.455,Z 524.694,A -85,B 0,C 180,E1 -526.068,E2 -526.068} C_VEL
LIN {X 0,Y 608.698,Z 531.408,A -85,B 0,C 180,E1 -526.159,E2 -526.159} C_VEL
LIN {X 0,Y 608.653,Z 569.876,A -85,B 0,C 180,E1 -526.648,E2 -526.648} C_VEL
LIN {X 0,Y 608.643,Z 585.329,A -85,B 0,C 180,E1 -526.987,E2 -526.987} C_VEL
LIN {X 0,Y 608.62,Z 600.184,A -85,B 0,C 180,E1 -527.453,E2 -527.453} C_VEL
LIN {X 0,Y 608.601,Z 613.655,A -85,B 0,C 180,E1 -528.003,E2 -528.003} C_VEL
LIN {X 0,Y 608.565,Z 628.083,A -85,B 0,C 180,E1 -528.743,E2 -528.743} C_VEL
LIN {X 0,Y 608.555,Z 641.677,A -85,B 0,C 180,E1 -529.604,E2 -529.604} C_VEL
LIN {X 0,Y 608.514,Z 653.748,A -85,B 0,C 180,E1 -530.527,E2 -530.527} C_VEL
LIN {X 0,Y 608.485,Z 664.795,A -85,B 0,C 180,E1 -531.531,E2 -531.531} C_VEL
LIN {X 0,Y 608.475,Z 675.547,A -85,B 0,C 180,E1 -532.7,E2 -532.7} C_VEL
LIN {X 0,Y 608.449,Z 684.517,A -85,B 0,C 180,E1 -533.866,E2 -533.866} C_VEL
LIN {X 0,Y 608.452,Z 691.964,A -85,B 0,C 180,E1 -535.03,E2 -535.03} C_VEL
LIN {X 0,Y 608.448,Z 698.939,A -85,B 0,C 180,E1 -536.357,E2 -536.357} C_VEL
LIN {X 0,Y 608.424,Z 704.438,A -85,B 0,C 180,E1 -537.683,E2 -537.683} C_VEL
LIN {X 0,Y 608.449,Z 707.728,A -85,B 0,C 180,E1 -538.676,E2 -538.676} C_VEL
LIN {X 0,Y 608.43,Z 710.961,A -85,B 0,C 180,E1 -540,E2 -540} C_VEL
LIN {X 0,Y 608.443,Z 713.003,A -85,B 0,C 180,E1 -541.323,E2 -541.323} C_VEL
LIN {X 0,Y 608.423,Z 713.913,A -85,B 0,C 180,E1 -542.648,E2 -542.648} C_VEL
LIN {X 0,Y 608.426,Z 713.691,A -85,B 0,C 180,E1 -543.974,E2 -543.974} C_VEL
LIN {X 0,Y 608.414,Z 712.336,A -85,B 0,C 180,E1 -545.302,E2 -545.302} C_VEL
LIN {X 0,Y 608.439,Z 709.788,A -85,B 0,C 180,E1 -546.633,E2 -546.633} C_VEL
LIN {X 0,Y 608.427,Z 705.976,A -85,B 0,C 180,E1 -547.967,E2 -547.967} C_VEL
LIN {X 0,Y 608.428,Z 700.673,A -85,B 0,C 180,E1 -549.347,E2 -549.347} C_VEL
LIN {X 0,Y 607.756,Z 698.396,A -85,B 0,C 180,E1 -549.857,E2 -549.857} C_VEL
LIN {X 0,Y 604.897,Z 694.438,A -85,B 0,C 180,E1 -550.674,E2 -550.674} C_VEL
LIN {X 0,Y 602.048,Z 690.027,A -85,B 0,C 180,E1 -551.475,E2 -551.475} C_VEL
LIN {X 0,Y 601.399,Z 687.007,A -85,B 0,C 180,E1 -551.957,E2 -551.957} C_VEL
LIN {X 0,Y 601.416,Z 678.277,A -85,B 0,C 180,E1 -553.172,E2 -553.172} C_VEL
LIN {X 0,Y 601.47,Z 667.845,A -85,B 0,C 180,E1 -554.377,E2 -554.377} C_VEL
LIN {X 0,Y 601.504,Z 657.121,A -85,B 0,C 180,E1 -555.415,E2 -555.415} C_VEL
LIN {X 0,Y 601.561,Z 644.793,A -85,B 0,C 180,E1 -556.416,E2 -556.416} C_VEL
LIN {X 0,Y 601.618,Z 632.594,A -85,B 0,C 180,E1 -557.243,E2 -557.243} C_VEL
LIN {X 0,Y 601.671,Z 618.439,A -85,B 0,C 180,E1 -558.031,E2 -558.031} C_VEL
LIN {X 0,Y 601.738,Z 604.245,A -85,B 0,C 180,E1 -558.664,E2 -558.664} C_VEL
LIN {X 0,Y 601.824,Z 589.406,A -85,B 0,C 180,E1 -559.174,E2 -559.174} C_VEL
LIN {X 0,Y 601.845,Z 574.245,A -85,B 0,C 180,E1 -559.55,E2 -559.55} C_VEL
LIN {X 0,Y 601.882,Z 557.007,A -85,B 0,C 180,E1 -559.815,E2 -559.815} C_VEL
LIN {X 0,Y 601.827,Z 527.166,A -85,B 0,C 180,E1 -560.181,E2 -560.181} C_VEL
LIN {X 0,Y 601.415,Z 525.569,A -85,B 0,C 180,E1 -560.232,E2 -560.232} C_VEL
LIN {X 0,Y 601.414,Z 525.564,A -85,B 0,C 180,E1 -562.683,E2 -562.683} C_VEL
LIN {X 0,Y 601.401,Z 525.565,A -85,B 0,C 180,E1 -564.878,E2 -564.878} C_VEL
LIN {X 0,Y 601.418,Z 525.572,A -85,B 0,C 180,E1 -567.867,E2 -567.867} C_VEL
LIN {X 0,Y 601.43,Z 525.571,A -85,B 0,C 180,E1 -570.164,E2 -570.164} C_VEL
LIN {X 0,Y 601.418,Z 525.565,A -85,B 0,C 180,E1 -572.714,E2 -572.714} C_VEL
LIN {X 0,Y 601.391,Z 525.566,A -85,B 0,C 180,E1 -575.111,E2 -575.111} C_VEL
LIN {X 0,Y 601.437,Z 525.561,A -85,B 0,C 180,E1 -577.418,E2 -577.418} C_VEL
LIN {X 0,Y 601.411,Z 525.571,A -85,B 0,C 180,E1 -579.995,E2 -579.995} C_VEL
LIN {X 0,Y 601.414,Z 525.568,A -85,B 0,C 180,E1 -582.67,E2 -582.67} C_VEL
LIN {X 0,Y 601.397,Z 525.566,A -85,B 0,C 180,E1 -585.467,E2 -585.467} C_VEL
LIN {X 0,Y 601.422,Z 525.574,A -85,B 0,C 180,E1 -588.407,E2 -588.407} C_VEL
LIN {X 0,Y 601.432,Z 525.565,A -85,B 0,C 180,E1 -590.875,E2 -590.875} C_VEL
LIN {X 0,Y 601.401,Z 525.565,A -85,B 0,C 180,E1 -593.417,E2 -593.417} C_VEL
LIN {X 0,Y 601.434,Z 525.564,A -85,B 0,C 180,E1 -596.064,E2 -596.064} C_VEL
LIN {X 0,Y 601.441,Z 525.571,A -85,B 0,C 180,E1 -598.541,E2 -598.541} C_VEL
LIN {X 0,Y 601.434,Z 525.562,A -85,B 0,C 180,E1 -601.373,E2 -601.373} C_VEL
LIN {X 0,Y 601.402,Z 525.565,A -85,B 0,C 180,E1 -603.636,E2 -603.636} C_VEL
LIN {X 0,Y 601.417,Z 525.572,A -85,B 0,C 180,E1 -606.589,E2 -606.589} C_VEL
LIN {X 0,Y 601.429,Z 525.562,A -85,B 0,C 180,E1 -609.478,E2 -609.478} C_VEL
LIN {X 0,Y 601.398,Z 525.568,A -85,B 0,C 180,E1 -612.311,E2 -612.311} C_VEL
LIN {X 0,Y 601.416,Z 525.567,A -85,B 0,C 180,E1 -614.408,E2 -614.408} C_VEL
LIN {X 0,Y 601.422,Z 525.569,A -85,B 0,C 180,E1 -617.172,E2 -617.172} C_VEL
LIN {X 0,Y 601.428,Z 525.562,A -85,B 0,C 180,E1 -619.905,E2 -619.905} C_VEL
LIN {X 0,Y 601.442,Z 525.564,A -85,B 0,C 180,E1 -622.615,E2 -622.615} C_VEL
LIN {X 0,Y 601.419,Z 525.569,A -85,B 0,C 180,E1 -625.308,E2 -625.308} C_VEL
LIN {X 0,Y 601.433,Z 525.561,A -85,B 0,C 180,E1 -627.991,E2 -627.991} C_VEL
LIN {X 0,Y 601.443,Z 525.563,A -85,B 0,C 180,E1 -630.669,E2 -630.669} C_VEL
LIN {X 0,Y 601.435,Z 525.569,A -85,B 0,C 180,E1 -633.349,E2 -633.349} C_VEL
LIN {X 0,Y 601.431,Z 525.562,A -85,B 0,C 180,E1 -636.036,E2 -636.036} C_VEL
LIN {X 0,Y 601.438,Z 525.561,A -85,B 0,C 180,E1 -638.06,E2 -638.06} C_VEL
LIN {X 0,Y 601.421,Z 525.568,A -85,B 0,C 180,E1 -641.012,E2 -641.012} C_VEL
LIN {X 0,Y 601.423,Z 525.571,A -85,B 0,C 180,E1 -643.515,E2 -643.515} C_VEL
LIN {X 0,Y 601.437,Z 525.561,A -85,B 0,C 180,E1 -646.286,E2 -646.286} C_VEL
LIN {X 0,Y 601.416,Z 525.567,A -85,B 0,C 180,E1 -649.098,E2 -649.098} C_VEL
LIN {X 0,Y 601.418,Z 525.567,A -85,B 0,C 180,E1 -651.958,E2 -651.958} C_VEL
LIN {X 0,Y 601.435,Z 525.562,A -85,B 0,C 180,E1 -654.293,E2 -654.293} C_VEL
LIN {X 0,Y 601.447,Z 525.562,A -85,B 0,C 180,E1 -657.111,E2 -657.111} C_VEL
LIN {X 0,Y 601.423,Z 525.568,A -85,B 0,C 180,E1 -659.392,E2 -659.392} C_VEL
LIN {X 0,Y 601.414,Z 525.575,A -85,B 0,C 180,E1 -661.726,E2 -661.726} C_VEL
LIN {X 0,Y 601.43,Z 525.566,A -85,B 0,C 180,E1 -664.118,E2 -664.118} C_VEL
LIN {X 0,Y 601.408,Z 525.565,A -85,B 0,C 180,E1 -666.582,E2 -666.582} C_VEL
LIN {X 0,Y 601.439,Z 525.565,A -85,B 0,C 180,E1 -669.536,E2 -669.536} C_VEL
LIN {X 0,Y 601.423,Z 525.571,A -85,B 0,C 180,E1 -671.765,E2 -671.765} C_VEL
LIN {X 0,Y 601.419,Z 525.565,A -85,B 0,C 180,E1 -674.535,E2 -674.535} C_VEL
LIN {X 0,Y 601.409,Z 525.565,A -85,B 0,C 180,E1 -677.33,E2 -677.33} C_VEL
LIN {X 0,Y 601.411,Z 525.574,A -85,B 0,C 180,E1 -680.005,E2 -680.005} C_VEL
LIN {X 0,Y 601.434,Z 525.564,A -85,B 0,C 180,E1 -682.617,E2 -682.617} C_VEL
LIN {X 0,Y 601.427,Z 525.562,A -85,B 0,C 180,E1 -685.069,E2 -685.069} C_VEL
LIN {X 0,Y 601.422,Z 525.563,A -85,B 0,C 180,E1 -687.484,E2 -687.484} C_VEL
LIN {X 0,Y 601.445,Z 525.564,A -85,B 0,C 180,E1 -689.848,E2 -689.848} C_VEL
LIN {X 0,Y 601.421,Z 525.569,A -85,B 0,C 180,E1 -691.973,E2 -691.973} C_VEL
LIN {X 0,Y 601.768,Z 528.895,A -85,B 0,C 180,E1 -692.032,E2 -692.032} C_VEL
LIN {X 0,Y 601.75,Z 589.105,A -85,B 0,C 180,E1 -692.778,E2 -692.778} C_VEL
LIN {X 0,Y 601.68,Z 603.266,A -85,B 0,C 180,E1 -693.088,E2 -693.088} C_VEL
LIN {X 0,Y 601.648,Z 616.519,A -85,B 0,C 180,E1 -693.508,E2 -693.508} C_VEL
LIN {X 0,Y 601.619,Z 628.747,A -85,B 0,C 180,E1 -694.018,E2 -694.018} C_VEL
LIN {X 0,Y 601.56,Z 641.076,A -85,B 0,C 180,E1 -694.667,E2 -694.667} C_VEL
LIN {X 0,Y 601.532,Z 653.113,A -85,B 0,C 180,E1 -695.452,E2 -695.452} C_VEL
LIN {X 0,Y 601.47,Z 664.035,A -85,B 0,C 180,E1 -696.318,E2 -696.318} C_VEL
LIN {X 0,Y 601.435,Z 674.471,A -85,B 0,C 180,E1 -697.318,E2 -697.318} C_VEL
LIN {X 0,Y 601.418,Z 683.817,A -85,B 0,C 180,E1 -698.402,E2 -698.402} C_VEL
LIN {X 0,Y 601.384,Z 691.453,A -85,B 0,C 180,E1 -699.477,E2 -699.477} C_VEL
LIN {X 0,Y 601.378,Z 697.694,A -85,B 0,C 180,E1 -700.545,E2 -700.545} C_VEL
LIN {X 0,Y 601.343,Z 702.756,A -85,B 0,C 180,E1 -701.606,E2 -701.606} C_VEL
LIN {X 0,Y 601.327,Z 706.793,A -85,B 0,C 180,E1 -702.661,E2 -702.661} C_VEL
LIN {X 0,Y 601.346,Z 709.86,A -85,B 0,C 180,E1 -703.711,E2 -703.711} C_VEL
LIN {X 0,Y 601.315,Z 712.6,A -85,B 0,C 180,E1 -705.101,E2 -705.101} C_VEL
LIN {X 0,Y 601.335,Z 713.878,A -85,B 0,C 180,E1 -706.483,E2 -706.483} C_VEL
LIN {X 0,Y 601.34,Z 713.736,A -85,B 0,C 180,E1 -707.856,E2 -707.856} C_VEL
LIN {X 0,Y 601.334,Z 712.224,A -85,B 0,C 180,E1 -709.223,E2 -709.223} C_VEL
LIN {X 0,Y 601.335,Z 709.314,A -85,B 0,C 180,E1 -710.583,E2 -710.583} C_VEL
LIN {X 0,Y 601.348,Z 704.957,A -85,B 0,C 180,E1 -711.938,E2 -711.938} C_VEL
LIN {X 0,Y 601.349,Z 699.041,A -85,B 0,C 180,E1 -713.289,E2 -713.289} C_VEL
LIN {X 0,Y 601.383,Z 692.391,A -85,B 0,C 180,E1 -714.468,E2 -714.468} C_VEL
LIN {X 0,Y 601.417,Z 684.165,A -85,B 0,C 180,E1 -715.644,E2 -715.644} C_VEL
LIN {X 0,Y 601.425,Z 675.643,A -85,B 0,C 180,E1 -716.651,E2 -716.651} C_VEL
LIN {X 0,Y 601.468,Z 665.362,A -85,B 0,C 180,E1 -717.656,E2 -717.656} C_VEL
LIN {X 0,Y 601.491,Z 653.947,A -85,B 0,C 180,E1 -718.578,E2 -718.578} C_VEL
LIN {X 0,Y 601.555,Z 642.583,A -85,B 0,C 180,E1 -719.331,E2 -719.331} C_VEL
LIN {X 0,Y 601.586,Z 630.2,A -85,B 0,C 180,E1 -720,E2 -720} C_VEL
LIN {X 0,Y 601.646,Z 617.515,A -85,B 0,C 180,E1 -720.544,E2 -720.544} C_VEL
LIN {X 0,Y 601.691,Z 603.235,A -85,B 0,C 180,E1 -721.004,E2 -721.004} C_VEL
LIN {X 0,Y 601.725,Z 588.847,A -85,B 0,C 180,E1 -721.318,E2 -721.318} C_VEL
LIN {X 0,Y 601.742,Z 526.995,A -85,B 0,C 180,E1 -722.081,E2 -722.081} C_VEL
LIN {X 0,Y 601.404,Z 525.57,A -85,B 0,C 180,E1 -722.114,E2 -722.114} C_VEL
LIN {X 0,Y 601.431,Z 525.562,A -85,B 0,C 180,E1 -724.692,E2 -724.692} C_VEL
LIN {X 0,Y 601.436,Z 525.568,A -85,B 0,C 180,E1 -727.385,E2 -727.385} C_VEL
LIN {X 0,Y 601.432,Z 525.565,A -85,B 0,C 180,E1 -730.095,E2 -730.095} C_VEL
LIN {X 0,Y 601.418,Z 525.565,A -85,B 0,C 180,E1 -732.828,E2 -732.828} C_VEL
LIN {X 0,Y 601.41,Z 525.575,A -85,B 0,C 180,E1 -735.592,E2 -735.592} C_VEL
LIN {X 0,Y 601.42,Z 525.564,A -85,B 0,C 180,E1 -738.392,E2 -738.392} C_VEL
LIN {X 0,Y 601.41,Z 525.571,A -85,B 0,C 180,E1 -741.239,E2 -741.239} C_VEL
LIN {X 0,Y 601.455,Z 525.56,A -85,B 0,C 180,E1 -744.141,E2 -744.141} C_VEL
LIN {X 0,Y 601.456,Z 525.564,A -85,B 0,C 180,E1 -747.111,E2 -747.111} C_VEL
LIN {X 0,Y 601.447,Z 525.56,A -85,B 0,C 180,E1 -750.163,E2 -750.163} C_VEL
LIN {X 0,Y 601.418,Z 525.565,A -85,B 0,C 180,E1 -752.716,E2 -752.716} C_VEL
LIN {X 0,Y 601.394,Z 525.573,A -85,B 0,C 180,E1 -755.113,E2 -755.113} C_VEL
LIN {X 0,Y 601.436,Z 525.57,A -85,B 0,C 180,E1 -757.419,E2 -757.419} C_VEL
LIN {X 0,Y 601.41,Z 525.565,A -85,B 0,C 180,E1 -759.995,E2 -759.995} C_VEL
LIN {X 0,Y 601.412,Z 525.567,A -85,B 0,C 180,E1 -762.671,E2 -762.671} C_VEL
LIN {X 0,Y 601.425,Z 525.568,A -85,B 0,C 180,E1 -765.483,E2 -765.483} C_VEL
LIN {X 0,Y 601.423,Z 525.564,A -85,B 0,C 180,E1 -768.407,E2 -768.407} C_VEL
LIN {X 0,Y 601.438,Z 525.568,A -85,B 0,C 180,E1 -770.876,E2 -770.876} C_VEL
LIN {X 0,Y 601.406,Z 525.57,A -85,B 0,C 180,E1 -773.418,E2 -773.418} C_VEL
LIN {X 0,Y 601.435,Z 525.562,A -85,B 0,C 180,E1 -776.064,E2 -776.064} C_VEL
LIN {X 0,Y 601.443,Z 525.565,A -85,B 0,C 180,E1 -778.542,E2 -778.542} C_VEL
LIN {X 0,Y 601.426,Z 525.597,A -85,B 0,C 180,E1 -779.788,E2 -779.788} C_VEL
LIN {X 0,Y 601.963,Z 528.605,A -85,B 0,C 180,E1 -780.252,E2 -780.252} C_VEL
LIN {X 0,Y 601.864,Z 548.654,A -85,B 0,C 180,E1 -783.097,E2 -783.097} C_VEL
LIN {X 0,Y 601.734,Z 568.704,A -85,B 0,C 180,E1 -785.872,E2 -785.872} C_VEL
LIN {X 0,Y 601.655,Z 588.753,A -85,B 0,C 180,E1 -788.591,E2 -788.591} C_VEL
LIN {X 0,Y 601.611,Z 609.669,A -85,B 0,C 180,E1 -791.376,E2 -791.376} C_VEL
LIN {X 0,Y 601.484,Z 631.525,A -85,B 0,C 180,E1 -794.237,E2 -794.237} C_VEL
LIN {X 0,Y 601.475,Z 651.491,A -85,B 0,C 180,E1 -796.819,E2 -796.819} C_VEL
LIN {X 0,Y 601.626,Z 673.644,A -85,B 0,C 180,E1 -797.091,E2 -797.091} C_VEL
LIN {X 0,Y 601.609,Z 759.97,A -85,B 0,C 180,E1 -798.14,E2 -798.14} C_VEL
LIN {X 0,Y 601.586,Z 773.232,A -85,B 0,C 180,E1 -798.439,E2 -798.439} C_VEL
LIN {X 0,Y 601.575,Z 785.668,A -85,B 0,C 180,E1 -798.855,E2 -798.855} C_VEL
LIN {X 0,Y 601.524,Z 797.642,A -85,B 0,C 180,E1 -799.397,E2 -799.397} C_VEL
LIN {X 0,Y 601.477,Z 809.204,A -85,B 0,C 180,E1 -800.076,E2 -800.076} C_VEL
LIN {X 0,Y 601.444,Z 819.599,A -85,B 0,C 180,E1 -800.839,E2 -800.839} C_VEL
LIN {X 0,Y 601.429,Z 828.116,A -85,B 0,C 180,E1 -801.601,E2 -801.601} C_VEL
LIN {X 0,Y 601.418,Z 835.964,A -85,B 0,C 180,E1 -802.446,E2 -802.446} C_VEL
LIN {X 0,Y 601.37,Z 843.227,A -85,B 0,C 180,E1 -803.398,E2 -803.398} C_VEL
LIN {X 0,Y 601.372,Z 848.868,A -85,B 0,C 180,E1 -804.299,E2 -804.299} C_VEL
LIN {X 0,Y 601.336,Z 853.952,A -85,B 0,C 180,E1 -805.308,E2 -805.308} C_VEL
LIN {X 0,Y 601.367,Z 857.897,A -85,B 0,C 180,E1 -806.315,E2 -806.315} C_VEL
LIN {X 0,Y 601.325,Z 860.81,A -85,B 0,C 180,E1 -807.321,E2 -807.321} C_VEL
LIN {X 0,Y 601.34,Z 862.203,A -85,B 0,C 180,E1 -807.991,E2 -807.991} C_VEL
LIN {X 0,Y 601.339,Z 863.784,A -85,B 0,C 180,E1 -809.331,E2 -809.331} C_VEL
LIN {X 0,Y 601.335,Z 864,A -85,B 0,C 180,E1 -810,E2 -810} C_VEL
LIN {X 0,Y 601.348,Z 863.184,A -85,B 0,C 180,E1 -811.34,E2 -811.34} C_VEL
LIN {X 0,Y 601.34,Z 862.201,A -85,B 0,C 180,E1 -812.01,E2 -812.01} C_VEL
LIN {X 0,Y 601.325,Z 860.808,A -85,B 0,C 180,E1 -812.68,E2 -812.68} C_VEL
LIN {X 0,Y 601.368,Z 857.895,A -85,B 0,C 180,E1 -813.686,E2 -813.686} C_VEL
LIN {X 0,Y 601.336,Z 853.948,A -85,B 0,C 180,E1 -814.693,E2 -814.693} C_VEL
LIN {X 0,Y 601.372,Z 847.874,A -85,B 0,C 180,E1 -815.87,E2 -815.87} C_VEL
LIN {X 0,Y 601.382,Z 841.233,A -85,B 0,C 180,E1 -816.88,E2 -816.88} C_VEL
LIN {X 0,Y 601.4,Z 832.986,A -85,B 0,C 180,E1 -817.893,E2 -817.893} C_VEL
LIN {X 0,Y 601.436,Z 824.532,A -85,B 0,C 180,E1 -818.738,E2 -818.738} C_VEL
LIN {X 0,Y 601.44,Z 814.087,A -85,B 0,C 180,E1 -819.586,E2 -819.586} C_VEL
LIN {X 0,Y 601.489,Z 803.75,A -85,B 0,C 180,E1 -820.264,E2 -820.264} C_VEL
LIN {X 0,Y 601.537,Z 792.896,A -85,B 0,C 180,E1 -820.836,E2 -820.836} C_VEL
LIN {X 0,Y 601.563,Z 780.369,A -85,B 0,C 180,E1 -821.341,E2 -821.341} C_VEL
LIN {X 0,Y 601.603,Z 767.339,A -85,B 0,C 180,E1 -821.711,E2 -821.711} C_VEL
LIN {X 0,Y 601.619,Z 754.056,A -85,B 0,C 180,E1 -821.946,E2 -821.946} C_VEL
LIN {X 0,Y 601.537,Z 652.112,A -85,B 0,C 180,E1 -823.169,E2 -823.169} C_VEL
LIN {X 0,Y 601.473,Z 651.234,A -85,B 0,C 180,E1 -823.214,E2 -823.214} C_VEL
LIN {X 0,Y 601.512,Z 630.182,A -85,B 0,C 180,E1 -825.937,E2 -825.937} C_VEL
LIN {X 0,Y 601.612,Z 609.664,A -85,B 0,C 180,E1 -828.624,E2 -828.624} C_VEL
LIN {X 0,Y 601.672,Z 587.41,A -85,B 0,C 180,E1 -831.589,E2 -831.589} C_VEL
LIN {X 0,Y 601.768,Z 566.991,A -85,B 0,C 180,E1 -834.362,E2 -834.362} C_VEL
LIN {X 0,Y 601.848,Z 547.311,A -85,B 0,C 180,E1 -837.092,E2 -837.092} C_VEL
LIN {X 0,Y 601.963,Z 528.598,A -85,B 0,C 180,E1 -839.749,E2 -839.749} C_VEL
LIN {X 0,Y 601.411,Z 525.571,A -85,B 0,C 180,E1 -840.238,E2 -840.238} C_VEL
LIN {X 0,Y 601.425,Z 525.569,A -85,B 0,C 180,E1 -842.715,E2 -842.715} C_VEL
LIN {X 0,Y 601.421,Z 525.571,A -85,B 0,C 180,E1 -845.115,E2 -845.115} C_VEL
LIN {X 0,Y 601.438,Z 525.564,A -85,B 0,C 180,E1 -847.419,E2 -847.419} C_VEL
LIN {X 0,Y 601.415,Z 525.564,A -85,B 0,C 180,E1 -849.995,E2 -849.995} C_VEL
LIN {X 0,Y 601.411,Z 525.573,A -85,B 0,C 180,E1 -852.671,E2 -852.671} C_VEL
LIN {X 0,Y 601.431,Z 525.563,A -85,B 0,C 180,E1 -855.482,E2 -855.482} C_VEL
LIN {X 0,Y 601.428,Z 525.568,A -85,B 0,C 180,E1 -858.407,E2 -858.407} C_VEL
LIN {X 0,Y 601.438,Z 525.568,A -85,B 0,C 180,E1 -860.875,E2 -860.875} C_VEL
LIN {X 0,Y 601.403,Z 525.566,A -85,B 0,C 180,E1 -863.417,E2 -863.417} C_VEL
LIN {X 0,Y 601.436,Z 525.564,A -85,B 0,C 180,E1 -866.064,E2 -866.064} C_VEL
LIN {X 0,Y 601.434,Z 525.565,A -85,B 0,C 180,E1 -869.059,E2 -869.059} C_VEL
LIN {X 0,Y 601.428,Z 525.563,A -85,B 0,C 180,E1 -871.373,E2 -871.373} C_VEL
LIN {X 0,Y 601.404,Z 525.566,A -85,B 0,C 180,E1 -873.636,E2 -873.636} C_VEL
LIN {X 0,Y 601.421,Z 525.572,A -85,B 0,C 180,E1 -876.589,E2 -876.589} C_VEL
LIN {X 0,Y 601.43,Z 525.563,A -85,B 0,C 180,E1 -879.478,E2 -879.478} C_VEL
LIN {X 0,Y 601.396,Z 525.577,A -85,B 0,C 180,E1 -882.311,E2 -882.311} C_VEL
LIN {X 0,Y 601.411,Z 525.575,A -85,B 0,C 180,E1 -884.408,E2 -884.408} C_VEL
LIN {X 0,Y 601.443,Z 525.565,A -85,B 0,C 180,E1 -885.873,E2 -885.873} C_VEL
LIN {X 0,Y 601.909,Z 528.164,A -85,B 0,C 180,E1 -885.923,E2 -885.923} C_VEL
LIN {X 0,Y 601.861,Z 569.055,A -85,B 0,C 180,E1 -886.443,E2 -886.443} C_VEL
LIN {X 0,Y 601.815,Z 584.358,A -85,B 0,C 180,E1 -886.772,E2 -886.772} C_VEL
LIN {X 0,Y 601.786,Z 600.003,A -85,B 0,C 180,E1 -887.265,E2 -887.265} C_VEL
LIN {X 0,Y 601.715,Z 614.456,A -85,B 0,C 180,E1 -887.863,E2 -887.863} C_VEL
LIN {X 0,Y 601.657,Z 628.856,A -85,B 0,C 180,E1 -888.62,E2 -888.62} C_VEL
LIN {X 0,Y 601.608,Z 642.181,A -85,B 0,C 180,E1 -889.482,E2 -889.482} C_VEL
LIN {X 0,Y 601.516,Z 654.178,A -85,B 0,C 180,E1 -890.416,E2 -890.416} C_VEL
LIN {X 0,Y 601.472,Z 665.158,A -85,B 0,C 180,E1 -891.432,E2 -891.432} C_VEL
LIN {X 0,Y 601.431,Z 675.844,A -85,B 0,C 180,E1 -892.614,E2 -892.614} C_VEL
LIN {X 0,Y 601.4,Z 684.675,A -85,B 0,C 180,E1 -893.781,E2 -893.781} C_VEL
LIN {X 0,Y 601.392,Z 692.183,A -85,B 0,C 180,E1 -894.971,E2 -894.971} C_VEL
LIN {X 0,Y 601.366,Z 699.116,A -85,B 0,C 180,E1 -896.314,E2 -896.314} C_VEL
LIN {X 0,Y 601.336,Z 704.574,A -85,B 0,C 180,E1 -897.655,E2 -897.655} C_VEL
LIN {X 0,Y 601.35,Z 707.829,A -85,B 0,C 180,E1 -898.66,E2 -898.66} C_VEL
LIN {X 0,Y 601.331,Z 711.038,A -85,B 0,C 180,E1 -900,E2 -900} C_VEL
LIN {X 0,Y 601.343,Z 713.049,A -85,B 0,C 180,E1 -901.339,E2 -901.339} C_VEL
LIN {X 0,Y 601.321,Z 713.924,A -85,B 0,C 180,E1 -902.679,E2 -902.679} C_VEL
LIN {X 0,Y 601.337,Z 713.669,A -85,B 0,C 180,E1 -904.021,E2 -904.021} C_VEL
LIN {X 0,Y 601.328,Z 712.281,A -85,B 0,C 180,E1 -905.365,E2 -905.365} C_VEL
LIN {X 0,Y 601.354,Z 709.706,A -85,B 0,C 180,E1 -906.711,E2 -906.711} C_VEL
LIN {X 0,Y 601.347,Z 705.863,A -85,B 0,C 180,E1 -908.062,E2 -908.062} C_VEL
LIN {X 0,Y 601.344,Z 700.702,A -85,B 0,C 180,E1 -909.417,E2 -909.417} C_VEL
LIN {X 0,Y 601.372,Z 694.072,A -85,B 0,C 180,E1 -910.777,E2 -910.777} C_VEL
LIN {X 0,Y 601.399,Z 687.007,A -85,B 0,C 180,E1 -911.957,E2 -911.957} C_VEL
LIN {X 0,Y 600.744,Z 683.899,A -85,B 0,C 180,E1 -912.43,E2 -912.43} C_VEL
LIN {X 0,Y 595.498,Z 674.199,A -85,B 0,C 180,E1 -913.779,E2 -913.779} C_VEL
LIN {X 0,Y 594.507,Z 670.548,A -85,B 0,C 180,E1 -914.219,E2 -914.219} C_VEL
LIN {X 0,Y 594.446,Z 669.246,A -85,B 0,C 180,E1 -914.363,E2 -914.363} C_VEL
LIN {X 0,Y 594.492,Z 658.658,A -85,B 0,C 180,E1 -915.426,E2 -915.426} C_VEL
LIN {X 0,Y 594.588,Z 647.235,A -85,B 0,C 180,E1 -916.391,E2 -916.391} C_VEL
LIN {X 0,Y 594.67,Z 634.811,A -85,B 0,C 180,E1 -917.273,E2 -917.273} C_VEL
LIN {X 0,Y 594.775,Z 621.211,A -85,B 0,C 180,E1 -918.069,E2 -918.069} C_VEL
LIN {X 0,Y 594.901,Z 606.712,A -85,B 0,C 180,E1 -918.749,E2 -918.749} C_VEL
LIN {X 0,Y 594.968,Z 592.758,A -85,B 0,C 180,E1 -919.261,E2 -919.261} C_VEL
LIN {X 0,Y 595.036,Z 577.748,A -85,B 0,C 180,E1 -919.67,E2 -919.67} C_VEL
LIN {X 0,Y 595.086,Z 562.677,A -85,B 0,C 180,E1 -919.938,E2 -919.938} C_VEL
LIN {X 0,Y 595.062,Z 528.717,A -85,B 0,C 180,E1 -920.363,E2 -920.363} C_VEL
LIN {X 0,Y 594.381,Z 526.444,A -85,B 0,C 180,E1 -920.414,E2 -920.414} C_VEL
LIN {X 0,Y 594.359,Z 526.443,A -85,B 0,C 180,E1 -922.967,E2 -922.967} C_VEL
LIN {X 0,Y 594.374,Z 526.442,A -85,B 0,C 180,E1 -925.193,E2 -925.193} C_VEL
LIN {X 0,Y 594.388,Z 526.442,A -85,B 0,C 180,E1 -927.526,E2 -927.526} C_VEL
LIN {X 0,Y 594.387,Z 526.445,A -85,B 0,C 180,E1 -930.328,E2 -930.328} C_VEL
LIN {X 0,Y 594.377,Z 526.44,A -85,B 0,C 180,E1 -932.95,E2 -932.95} C_VEL
LIN {X 0,Y 594.349,Z 526.444,A -85,B 0,C 180,E1 -935.409,E2 -935.409} C_VEL
LIN {X 0,Y 594.39,Z 526.445,A -85,B 0,C 180,E1 -937.94,E2 -937.94} C_VEL
LIN {X 0,Y 594.378,Z 526.442,A -85,B 0,C 180,E1 -940.822,E2 -940.822} C_VEL
LIN {X 0,Y 594.383,Z 526.443,A -85,B 0,C 180,E1 -943.841,E2 -943.841} C_VEL
LIN {X 0,Y 594.365,Z 526.446,A -85,B 0,C 180,E1 -946.7,E2 -946.7} C_VEL
LIN {X 0,Y 594.367,Z 526.441,A -85,B 0,C 180,E1 -949.432,E2 -949.432} C_VEL
LIN {X 0,Y 594.388,Z 526.449,A -85,B 0,C 180,E1 -952.391,E2 -952.391} C_VEL
LIN {X 0,Y 594.393,Z 526.438,A -85,B 0,C 180,E1 -955.421,E2 -955.421} C_VEL
LIN {X 0,Y 594.392,Z 526.445,A -85,B 0,C 180,E1 -958.355,E2 -958.355} C_VEL
LIN {X 0,Y 594.384,Z 526.443,A -85,B 0,C 180,E1 -961.041,E2 -961.041} C_VEL
LIN {X 0,Y 594.384,Z 526.44,A -85,B 0,C 180,E1 -963.977,E2 -963.977} C_VEL
LIN {X 0,Y 594.387,Z 526.443,A -85,B 0,C 180,E1 -966.296,E2 -966.296} C_VEL
LIN {X 0,Y 594.403,Z 526.44,A -85,B 0,C 180,E1 -969.224,E2 -969.224} C_VEL
LIN {X 0,Y 594.354,Z 526.444,A -85,B 0,C 180,E1 -972.095,E2 -972.095} C_VEL
LIN {X 0,Y 594.369,Z 526.443,A -85,B 0,C 180,E1 -974.219,E2 -974.219} C_VEL
LIN {X 0,Y 594.371,Z 526.45,A -85,B 0,C 180,E1 -977.017,E2 -977.017} C_VEL
LIN {X 0,Y 594.389,Z 526.439,A -85,B 0,C 180,E1 -979.784,E2 -979.784} C_VEL
LIN {X 0,Y 594.394,Z 526.441,A -85,B 0,C 180,E1 -982.526,E2 -982.526} C_VEL
LIN {X 0,Y 594.389,Z 526.446,A -85,B 0,C 180,E1 -985.252,E2 -985.252} C_VEL
LIN {X 0,Y 594.402,Z 526.437,A -85,B 0,C 180,E1 -987.967,E2 -987.967} C_VEL
LIN {X 0,Y 594.415,Z 526.438,A -85,B 0,C 180,E1 -990.677,E2 -990.677} C_VEL
LIN {X 0,Y 594.387,Z 526.447,A -85,B 0,C 180,E1 -993.389,E2 -993.389} C_VEL
LIN {X 0,Y 594.38,Z 526.44,A -85,B 0,C 180,E1 -996.108,E2 -996.108} C_VEL
LIN {X 0,Y 594.381,Z 526.443,A -85,B 0,C 180,E1 -998.842,E2 -998.842} C_VEL
LIN {X 0,Y 594.394,Z 526.445,A -85,B 0,C 180,E1 -1001.595,E2 -1001.595} C_VEL
LIN {X 0,Y 594.387,Z 526.439,A -85,B 0,C 180,E1 -1004.377,E2 -1004.377} C_VEL
LIN {X 0,Y 594.39,Z 526.445,A -85,B 0,C 180,E1 -1007.193,E2 -1007.193} C_VEL
LIN {X 0,Y 594.375,Z 526.443,A -85,B 0,C 180,E1 -1010.053,E2 -1010.053} C_VEL
LIN {X 0,Y 594.361,Z 526.444,A -85,B 0,C 180,E1 -1012.967,E2 -1012.967} C_VEL
LIN {X 0,Y 594.376,Z 526.444,A -85,B 0,C 180,E1 -1015.193,E2 -1015.193} C_VEL
LIN {X 0,Y 594.381,Z 526.448,A -85,B 0,C 180,E1 -1017.526,E2 -1017.526} C_VEL
LIN {X 0,Y 594.397,Z 526.439,A -85,B 0,C 180,E1 -1020.33,E2 -1020.33} C_VEL
LIN {X 0,Y 594.376,Z 526.441,A -85,B 0,C 180,E1 -1022.95,E2 -1022.95} C_VEL
LIN {X 0,Y 594.38,Z 526.444,A -85,B 0,C 180,E1 -1025.406,E2 -1025.406} C_VEL
LIN {X 0,Y 594.383,Z 526.449,A -85,B 0,C 180,E1 -1027.94,E2 -1027.94} C_VEL
LIN {X 0,Y 594.383,Z 526.439,A -85,B 0,C 180,E1 -1030.823,E2 -1030.823} C_VEL
LIN {X 0,Y 594.363,Z 526.451,A -85,B 0,C 180,E1 -1033.84,E2 -1033.84} C_VEL
LIN {X 0,Y 594.376,Z 526.441,A -85,B 0,C 180,E1 -1036.702,E2 -1036.702} C_VEL
LIN {X 0,Y 594.37,Z 526.443,A -85,B 0,C 180,E1 -1039.434,E2 -1039.434} C_VEL
LIN {X 0,Y 594.389,Z 526.445,A -85,B 0,C 180,E1 -1042.391,E2 -1042.391} C_VEL
LIN {X 0,Y 594.378,Z 526.443,A -85,B 0,C 180,E1 -1044.672,E2 -1044.672} C_VEL
LIN {X 0,Y 594.374,Z 526.441,A -85,B 0,C 180,E1 -1047.088,E2 -1047.088} C_VEL
LIN {X 0,Y 594.397,Z 526.44,A -85,B 0,C 180,E1 -1049.669,E2 -1049.669} C_VEL
LIN {X 0,Y 594.399,Z 526.585,A -85,B 0,C 180,E1 -1051.813,E2 -1051.813} C_VEL
LIN {X 0,Y 594.926,Z 529.384,A -85,B 0,C 180,E1 -1051.861,E2 -1051.861} C_VEL
LIN {X 0,Y 594.876,Z 589.262,A -85,B 0,C 180,E1 -1052.612,E2 -1052.612} C_VEL
LIN {X 0,Y 594.793,Z 603.041,A -85,B 0,C 180,E1 -1052.917,E2 -1052.917} C_VEL
LIN {X 0,Y 594.738,Z 616.871,A -85,B 0,C 180,E1 -1053.362,E2 -1053.362} C_VEL
LIN {X 0,Y 594.678,Z 629.87,A -85,B 0,C 180,E1 -1053.919,E2 -1053.919} C_VEL
LIN {X 0,Y 594.593,Z 642.882,A -85,B 0,C 180,E1 -1054.63,E2 -1054.63} C_VEL
LIN {X 0,Y 594.514,Z 655.302,A -85,B 0,C 180,E1 -1055.476,E2 -1055.476} C_VEL
LIN {X 0,Y 594.43,Z 666.278,A -85,B 0,C 180,E1 -1056.39,E2 -1056.39} C_VEL
LIN {X 0,Y 594.382,Z 675.011,A -85,B 0,C 180,E1 -1057.259,E2 -1057.259} C_VEL
LIN {X 0,Y 594.354,Z 683.944,A -85,B 0,C 180,E1 -1058.314,E2 -1058.314} C_VEL
LIN {X 0,Y 594.306,Z 692.676,A -85,B 0,C 180,E1 -1059.583,E2 -1059.583} C_VEL
LIN {X 0,Y 594.294,Z 698.713,A -85,B 0,C 180,E1 -1060.663,E2 -1060.663} C_VEL
LIN {X 0,Y 594.255,Z 703.571,A -85,B 0,C 180,E1 -1061.736,E2 -1061.736} C_VEL
LIN {X 0,Y 594.247,Z 707.395,A -85,B 0,C 180,E1 -1062.803,E2 -1062.803} C_VEL
LIN {X 0,Y 594.244,Z 709.445,A -85,B 0,C 180,E1 -1063.511,E2 -1063.511} C_VEL
LIN {X 0,Y 594.227,Z 712.351,A -85,B 0,C 180,E1 -1064.919,E2 -1064.919} C_VEL
LIN {X 0,Y 594.251,Z 713.788,A -85,B 0,C 180,E1 -1066.318,E2 -1066.318} C_VEL
LIN {X 0,Y 594.236,Z 713.839,A -85,B 0,C 180,E1 -1067.709,E2 -1067.709} C_VEL
LIN {X 0,Y 594.233,Z 712.478,A -85,B 0,C 180,E1 -1069.092,E2 -1069.092} C_VEL
LIN {X 0,Y 594.254,Z 709.717,A -85,B 0,C 180,E1 -1070.47,E2 -1070.47} C_VEL
LIN {X 0,Y 594.277,Z 705.518,A -85,B 0,C 180,E1 -1071.842,E2 -1071.842} C_VEL
LIN {X 0,Y 594.27,Z 699.777,A -85,B 0,C 180,E1 -1073.208,E2 -1073.208} C_VEL
LIN {X 0,Y 594.308,Z 693.318,A -85,B 0,C 180,E1 -1074.402,E2 -1074.402} C_VEL
LIN {X 0,Y 594.364,Z 685.328,A -85,B 0,C 180,E1 -1075.592,E2 -1075.592} C_VEL
LIN {X 0,Y 594.405,Z 675.498,A -85,B 0,C 180,E1 -1076.781,E2 -1076.781} C_VEL
LIN {X 0,Y 594.454,Z 665.196,A -85,B 0,C 180,E1 -1077.798,E2 -1077.798} C_VEL
LIN {X 0,Y 594.505,Z 653.745,A -85,B 0,C 180,E1 -1078.73,E2 -1078.73} C_VEL
LIN {X 0,Y 594.588,Z 642.331,A -85,B 0,C 180,E1 -1079.492,E2 -1079.492} C_VEL
LIN {X 0,Y 594.647,Z 629.882,A -85,B 0,C 180,E1 -1080.17,E2 -1080.17} C_VEL
LIN {X 0,Y 594.746,Z 616.017,A -85,B 0,C 180,E1 -1080.762,E2 -1080.762} C_VEL
LIN {X 0,Y 594.813,Z 601.837,A -85,B 0,C 180,E1 -1081.206,E2 -1081.206} C_VEL
LIN {X 0,Y 594.846,Z 587.81,A -85,B 0,C 180,E1 -1081.502,E2 -1081.502} C_VEL
LIN {X 0,Y 594.878,Z 528.304,A -85,B 0,C 180,E1 -1082.243,E2 -1082.243} C_VEL
LIN {X 0,Y 594.376,Z 526.444,A -85,B 0,C 180,E1 -1082.287,E2 -1082.287} C_VEL
LIN {X 0,Y 594.399,Z 526.439,A -85,B 0,C 180,E1 -1084.748,E2 -1084.748} C_VEL
LIN {X 0,Y 594.389,Z 526.447,A -85,B 0,C 180,E1 -1087.474,E2 -1087.474} C_VEL
LIN {X 0,Y 594.392,Z 526.441,A -85,B 0,C 180,E1 -1090.216,E2 -1090.216} C_VEL
LIN {X 0,Y 594.365,Z 526.444,A -85,B 0,C 180,E1 -1092.983,E2 -1092.983} C_VEL
LIN {X 0,Y 594.363,Z 526.45,A -85,B 0,C 180,E1 -1095.781,E2 -1095.781} C_VEL
LIN {X 0,Y 594.384,Z 526.44,A -85,B 0,C 180,E1 -1098.618,E2 -1098.618} C_VEL
LIN {X 0,Y 594.368,Z 526.452,A -85,B 0,C 180,E1 -1101.504,E2 -1101.504} C_VEL
LIN {X 0,Y 594.386,Z 526.44,A -85,B 0,C 180,E1 -1104.446,E2 -1104.446} C_VEL
LIN {X 0,Y 594.387,Z 526.44,A -85,B 0,C 180,E1 -1106.7,E2 -1106.7} C_VEL
LIN {X 0,Y 594.38,Z 526.444,A -85,B 0,C 180,E1 -1108.999,E2 -1108.999} C_VEL
LIN {X 0,Y 594.391,Z 526.444,A -85,B 0,C 180,E1 -1111.646,E2 -1111.646} C_VEL
LIN {X 0,Y 594.378,Z 526.441,A -85,B 0,C 180,E1 -1114.58,E2 -1114.58} C_VEL
LIN {X 0,Y 594.391,Z 526.444,A -85,B 0,C 180,E1 -1117.609,E2 -1117.609} C_VEL
LIN {X 0,Y 594.37,Z 526.443,A -85,B 0,C 180,E1 -1120.567,E2 -1120.567} C_VEL
LIN {X 0,Y 594.379,Z 526.45,A -85,B 0,C 180,E1 -1123.299,E2 -1123.299} C_VEL
LIN {X 0,Y 594.366,Z 526.442,A -85,B 0,C 180,E1 -1126.161,E2 -1126.161} C_VEL
LIN {X 0,Y 594.377,Z 526.451,A -85,B 0,C 180,E1 -1129.178,E2 -1129.178} C_VEL
LIN {X 0,Y 594.384,Z 526.44,A -85,B 0,C 180,E1 -1132.06,E2 -1132.06} C_VEL
LIN {X 0,Y 594.385,Z 526.444,A -85,B 0,C 180,E1 -1134.672,E2 -1134.672} C_VEL
LIN {X 0,Y 594.381,Z 526.451,A -85,B 0,C 180,E1 -1137.089,E2 -1137.089} C_VEL
LIN {X 0,Y 594.419,Z 526.638,A -85,B 0,C 180,E1 -1139.553,E2 -1139.553} C_VEL
LIN {X 0,Y 595.203,Z 531.278,A -85,B 0,C 180,E1 -1140.27,E2 -1140.27} C_VEL
LIN {X 0,Y 595.032,Z 551.327,A -85,B 0,C 180,E1 -1143.143,E2 -1143.143} C_VEL
LIN {X 0,Y 594.86,Z 571.377,A -85,B 0,C 180,E1 -1145.946,E2 -1145.946} C_VEL
LIN {X 0,Y 594.742,Z 591.2,A -85,B 0,C 180,E1 -1148.662,E2 -1148.662} C_VEL
LIN {X 0,Y 594.628,Z 611.476,A -85,B 0,C 180,E1 -1151.391,E2 -1151.391} C_VEL
LIN {X 0,Y 594.518,Z 631.525,A -85,B 0,C 180,E1 -1154.048,E2 -1154.048} C_VEL
LIN {X 0,Y 594.469,Z 651.408,A -85,B 0,C 180,E1 -1156.65,E2 -1156.65} C_VEL
LIN {X 0,Y 594.765,Z 657.546,A -85,B 0,C 180,E1 -1156.744,E2 -1156.744} C_VEL
LIN {X 0,Y 594.662,Z 759.97,A -85,B 0,C 180,E1 -1157.999,E2 -1157.999} C_VEL
LIN {X 0,Y 594.629,Z 773.232,A -85,B 0,C 180,E1 -1158.301,E2 -1158.301} C_VEL
LIN {X 0,Y 594.607,Z 785.277,A -85,B 0,C 180,E1 -1158.708,E2 -1158.708} C_VEL
LIN {X 0,Y 594.538,Z 797.641,A -85,B 0,C 180,E1 -1159.271,E2 -1159.271} C_VEL
LIN {X 0,Y 594.472,Z 809.205,A -85,B 0,C 180,E1 -1159.958,E2 -1159.958} C_VEL
LIN {X 0,Y 594.413,Z 819.6,A -85,B 0,C 180,E1 -1160.73,E2 -1160.73} C_VEL
LIN {X 0,Y 594.383,Z 828.117,A -85,B 0,C 180,E1 -1161.501,E2 -1161.501} C_VEL
LIN {X 0,Y 594.347,Z 835.964,A -85,B 0,C 180,E1 -1162.356,E2 -1162.356} C_VEL
LIN {X 0,Y 594.282,Z 843.815,A -85,B 0,C 180,E1 -1163.409,E2 -1163.409} C_VEL
LIN {X 0,Y 594.289,Z 850.683,A -85,B 0,C 180,E1 -1164.572,E2 -1164.572} C_VEL
LIN {X 0,Y 594.271,Z 855.372,A -85,B 0,C 180,E1 -1165.592,E2 -1165.592} C_VEL
LIN {X 0,Y 594.268,Z 858.958,A -85,B 0,C 180,E1 -1166.61,E2 -1166.61} C_VEL
LIN {X 0,Y 594.226,Z 860.811,A -85,B 0,C 180,E1 -1167.289,E2 -1167.289} C_VEL
LIN {X 0,Y 594.239,Z 862.203,A -85,B 0,C 180,E1 -1167.967,E2 -1167.967} C_VEL
LIN {X 0,Y 594.239,Z 863.784,A -85,B 0,C 180,E1 -1169.323,E2 -1169.323} C_VEL
LIN {X 0,Y 594.236,Z 864,A -85,B 0,C 180,E1 -1170,E2 -1170} C_VEL
LIN {X 0,Y 594.247,Z 863.184,A -85,B 0,C 180,E1 -1171.356,E2 -1171.356} C_VEL
LIN {X 0,Y 594.239,Z 862.201,A -85,B 0,C 180,E1 -1172.034,E2 -1172.034} C_VEL
LIN {X 0,Y 594.226,Z 860.808,A -85,B 0,C 180,E1 -1172.712,E2 -1172.712} C_VEL
LIN {X 0,Y 594.289,Z 857.895,A -85,B 0,C 180,E1 -1173.73,E2 -1173.73} C_VEL
LIN {X 0,Y 594.241,Z 853.948,A -85,B 0,C 180,E1 -1174.749,E2 -1174.749} C_VEL
LIN {X 0,Y 594.304,Z 847.875,A -85,B 0,C 180,E1 -1175.94,E2 -1175.94} C_VEL
LIN {X 0,Y 594.309,Z 841.233,A -85,B 0,C 180,E1 -1176.962,E2 -1176.962} C_VEL
LIN {X 0,Y 594.359,Z 832.987,A -85,B 0,C 180,E1 -1177.987,E2 -1177.987} C_VEL
LIN {X 0,Y 594.382,Z 824.532,A -85,B 0,C 180,E1 -1178.843,E2 -1178.843} C_VEL
LIN {X 0,Y 594.423,Z 814.088,A -85,B 0,C 180,E1 -1179.7,E2 -1179.7} C_VEL
LIN {X 0,Y 594.489,Z 803.752,A -85,B 0,C 180,E1 -1180.387,E2 -1180.387} C_VEL
LIN {X 0,Y 594.56,Z 792.699,A -85,B 0,C 180,E1 -1180.974,E2 -1180.974} C_VEL
LIN {X 0,Y 594.598,Z 780.697,A -85,B 0,C 180,E1 -1181.464,E2 -1181.464} C_VEL
LIN {X 0,Y 594.645,Z 767.339,A -85,B 0,C 180,E1 -1181.85,E2 -1181.85} C_VEL
LIN {X 0,Y 594.693,Z 754.056,A -85,B 0,C 180,E1 -1182.087,E2 -1182.087} C_VEL
LIN {X 0,Y 594.656,Z 652.894,A -85,B 0,C 180,E1 -1183.315,E2 -1183.315} C_VEL
LIN {X 0,Y 594.464,Z 651.234,A -85,B 0,C 180,E1 -1183.373,E2 -1183.373} C_VEL
LIN {X 0,Y 594.568,Z 627.509,A -85,B 0,C 180,E1 -1186.481,E2 -1186.481} C_VEL
LIN {X 0,Y 594.672,Z 606.123,A -85,B 0,C 180,E1 -1189.324,E2 -1189.324} C_VEL
LIN {X 0,Y 594.809,Z 583.617,A -85,B 0,C 180,E1 -1192.37,E2 -1192.37} C_VEL
LIN {X 0,Y 594.917,Z 562.014,A -85,B 0,C 180,E1 -1195.356,E2 -1195.356} C_VEL
LIN {X 0,Y 595.097,Z 543.121,A -85,B 0,C 180,E1 -1198.024,E2 -1198.024} C_VEL
LIN {X 0,Y 595.158,Z 530.08,A -85,B 0,C 180,E1 -1199.907,E2 -1199.907} C_VEL
LIN {X 0,Y 594.391,Z 526.446,A -85,B 0,C 180,E1 -1200.485,E2 -1200.485} C_VEL
LIN {X 0,Y 594.383,Z 526.451,A -85,B 0,C 180,E1 -1202.95,E2 -1202.95} C_VEL
LIN {X 0,Y 594.362,Z 526.446,A -85,B 0,C 180,E1 -1205.409,E2 -1205.409} C_VEL
LIN {X 0,Y 594.386,Z 526.44,A -85,B 0,C 180,E1 -1207.941,E2 -1207.941} C_VEL
LIN {X 0,Y 594.378,Z 526.451,A -85,B 0,C 180,E1 -1210.822,E2 -1210.822} C_VEL
LIN {X 0,Y 594.369,Z 526.445,A -85,B 0,C 180,E1 -1213.3,E2 -1213.3} C_VEL
LIN {X 0,Y 594.373,Z 526.443,A -85,B 0,C 180,E1 -1216.16,E2 -1216.16} C_VEL
LIN {X 0,Y 594.385,Z 526.447,A -85,B 0,C 180,E1 -1218.536,E2 -1218.536} C_VEL
LIN {X 0,Y 594.391,Z 526.441,A -85,B 0,C 180,E1 -1221.295,E2 -1221.295} C_VEL
LIN {X 0,Y 594.354,Z 526.444,A -85,B 0,C 180,E1 -1223.755,E2 -1223.755} C_VEL
LIN {X 0,Y 594.383,Z 526.445,A -85,B 0,C 180,E1 -1226.239,E2 -1226.239} C_VEL
LIN {X 0,Y 594.394,Z 526.448,A -85,B 0,C 180,E1 -1228.651,E2 -1228.651} C_VEL
LIN {X 0,Y 594.386,Z 526.443,A -85,B 0,C 180,E1 -1231.042,E2 -1231.042} C_VEL
LIN {X 0,Y 594.391,Z 526.442,A -85,B 0,C 180,E1 -1233.977,E2 -1233.977} C_VEL
LIN {X 0,Y 594.39,Z 526.447,A -85,B 0,C 180,E1 -1236.296,E2 -1236.296} C_VEL
LIN {X 0,Y 594.404,Z 526.438,A -85,B 0,C 180,E1 -1239.224,E2 -1239.224} C_VEL
LIN {X 0,Y 594.354,Z 526.45,A -85,B 0,C 180,E1 -1242.095,E2 -1242.095} C_VEL
LIN {X 0,Y 594.364,Z 526.452,A -85,B 0,C 180,E1 -1244.219,E2 -1244.219} C_VEL
LIN {X 0,Y 594.372,Z 526.448,A -85,B 0,C 180,E1 -1245.678,E2 -1245.678} C_VEL
LIN {X 0,Y 595.146,Z 529.68,A -85,B 0,C 180,E1 -1245.742,E2 -1245.742} C_VEL
LIN {X 0,Y 595.066,Z 569.068,A -85,B 0,C 180,E1 -1246.249,E2 -1246.249} C_VEL
LIN {X 0,Y 594.994,Z 584.924,A -85,B 0,C 180,E1 -1246.596,E2 -1246.596} C_VEL
LIN {X 0,Y 594.92,Z 599.828,A -85,B 0,C 180,E1 -1247.072,E2 -1247.072} C_VEL
LIN {X 0,Y 594.856,Z 613.389,A -85,B 0,C 180,E1 -1247.635,E2 -1247.635} C_VEL
LIN {X 0,Y 594.774,Z 626.707,A -85,B 0,C 180,E1 -1248.325,E2 -1248.325} C_VEL
LIN {X 0,Y 594.64,Z 640.267,A -85,B 0,C 180,E1 -1249.185,E2 -1249.185} C_VEL
LIN {X 0,Y 594.557,Z 652.586,A -85,B 0,C 180,E1 -1250.131,E2 -1250.131} C_VEL
LIN {X 0,Y 594.47,Z 663.81,A -85,B 0,C 180,E1 -1251.159,E2 -1251.159} C_VEL
LIN {X 0,Y 594.399,Z 674.755,A -85,B 0,C 180,E1 -1252.356,E2 -1252.356} C_VEL
LIN {X 0,Y 594.371,Z 684.017,A -85,B 0,C 180,E1 -1253.576,E2 -1253.576} C_VEL
LIN {X 0,Y 594.335,Z 692.399,A -85,B 0,C 180,E1 -1254.912,E2 -1254.912} C_VEL
LIN {X 0,Y 594.287,Z 699.287,A -85,B 0,C 180,E1 -1256.27,E2 -1256.27} C_VEL
LIN {X 0,Y 594.251,Z 704.71,A -85,B 0,C 180,E1 -1257.627,E2 -1257.627} C_VEL
LIN {X 0,Y 594.253,Z 707.929,A -85,B 0,C 180,E1 -1258.644,E2 -1258.644} C_VEL
LIN {X 0,Y 594.232,Z 711.115,A -85,B 0,C 180,E1 -1260,E2 -1260} C_VEL
LIN {X 0,Y 594.243,Z 713.094,A -85,B 0,C 180,E1 -1261.355,E2 -1261.355} C_VEL
LIN {X 0,Y 594.222,Z 713.934,A -85,B 0,C 180,E1 -1262.711,E2 -1262.711} C_VEL
LIN {X 0,Y 594.25,Z 713.646,A -85,B 0,C 180,E1 -1264.069,E2 -1264.069} C_VEL
LIN {X 0,Y 594.244,Z 712.225,A -85,B 0,C 180,E1 -1265.429,E2 -1265.429} C_VEL
LIN {X 0,Y 594.271,Z 709.622,A -85,B 0,C 180,E1 -1266.792,E2 -1266.792} C_VEL
LIN {X 0,Y 594.278,Z 705.75,A -85,B 0,C 180,E1 -1268.158,E2 -1268.158} C_VEL
LIN {X 0,Y 594.266,Z 700.551,A -85,B 0,C 180,E1 -1269.53,E2 -1269.53} C_VEL
LIN {X 0,Y 594.317,Z 693.878,A -85,B 0,C 180,E1 -1270.906,E2 -1270.906} C_VEL
LIN {X 0,Y 594.335,Z 686.671,A -85,B 0,C 180,E1 -1272.116,E2 -1272.116} C_VEL
LIN {X 0,Y 594.393,Z 677.986,A -85,B 0,C 180,E1 -1273.33,E2 -1273.33} C_VEL
LIN {X 0,Y 594.446,Z 669.246,A -85,B 0,C 180,E1 -1274.363,E2 -1274.363} C_VEL
LIN {X 0,Y 593.848,Z 665.385,A -85,B 0,C 180,E1 -1274.791,E2 -1274.791} C_VEL
LIN {X 0,Y 591.076,Z 659.03,A -85,B 0,C 180,E1 -1275.477,E2 -1275.477} C_VEL
LIN {X 0,Y 588.272,Z 652.296,A -85,B 0,C 180,E1 -1276.131,E2 -1276.131} C_VEL
LIN {X 0,Y 587.624,Z 647.84,A -85,B 0,C 180,E1 -1276.505,E2 -1276.505} C_VEL
LIN {X 0,Y 587.737,Z 634.22,A -85,B 0,C 180,E1 -1277.484,E2 -1277.484} C_VEL
LIN {X 0,Y 587.868,Z 620.455,A -85,B 0,C 180,E1 -1278.289,E2 -1278.289} C_VEL
LIN {X 0,Y 588.039,Z 605.336,A -85,B 0,C 180,E1 -1278.994,E2 -1278.994} C_VEL
LIN {X 0,Y 588.175,Z 591.795,A -85,B 0,C 180,E1 -1279.484,E2 -1279.484} C_VEL
LIN {X 0,Y 588.265,Z 577.016,A -85,B 0,C 180,E1 -1279.884,E2 -1279.884} C_VEL
LIN {X 0,Y 588.284,Z 561.572,A -85,B 0,C 180,E1 -1280.156,E2 -1280.156} C_VEL
LIN {X 0,Y 588.286,Z 530.299,A -85,B 0,C 180,E1 -1280.549,E2 -1280.549} C_VEL
LIN {X 0,Y 587.373,Z 527.315,A -85,B 0,C 180,E1 -1280.623,E2 -1280.623} C_VEL
LIN {X 0,Y 587.317,Z 527.322,A -85,B 0,C 180,E1 -1283.259,E2 -1283.259} C_VEL
LIN {X 0,Y 587.333,Z 527.322,A -85,B 0,C 180,E1 -1285.516,E2 -1285.516} C_VEL
LIN {X 0,Y 587.35,Z 527.324,A -85,B 0,C 180,E1 -1287.817,E2 -1287.817} C_VEL
LIN {X 0,Y 587.338,Z 527.32,A -85,B 0,C 180,E1 -1290.509,E2 -1290.509} C_VEL
LIN {X 0,Y 587.334,Z 527.318,A -85,B 0,C 180,E1 -1293.396,E2 -1293.396} C_VEL
LIN {X 0,Y 587.291,Z 527.329,A -85,B 0,C 180,E1 -1295.9,E2 -1295.9} C_VEL
LIN {X 0,Y 587.335,Z 527.323,A -85,B 0,C 180,E1 -1298.479,E2 -1298.479} C_VEL
LIN {X 0,Y 587.337,Z 527.317,A -85,B 0,C 180,E1 -1301.156,E2 -1301.156} C_VEL
LIN {X 0,Y 587.335,Z 527.325,A -85,B 0,C 180,E1 -1304.114,E2 -1304.114} C_VEL
LIN {X 0,Y 587.313,Z 527.322,A -85,B 0,C 180,E1 -1306.993,E2 -1306.993} C_VEL
LIN {X 0,Y 587.317,Z 527.321,A -85,B 0,C 180,E1 -1309.745,E2 -1309.745} C_VEL
LIN {X 0,Y 587.343,Z 527.326,A -85,B 0,C 180,E1 -1312.392,E2 -1312.392} C_VEL
LIN {X 0,Y 587.354,Z 527.315,A -85,B 0,C 180,E1 -1315.651,E2 -1315.651} C_VEL
LIN {X 0,Y 587.353,Z 527.32,A -85,B 0,C 180,E1 -1318.231,E2 -1318.231} C_VEL
LIN {X 0,Y 587.35,Z 527.322,A -85,B 0,C 180,E1 -1320.866,E2 -1320.866} C_VEL
LIN {X 0,Y 587.358,Z 527.315,A -85,B 0,C 180,E1 -1323.819,E2 -1323.819} C_VEL
LIN {X 0,Y 587.335,Z 527.318,A -85,B 0,C 180,E1 -1325.993,E2 -1325.993} C_VEL
LIN {X 0,Y 587.323,Z 527.321,A -85,B 0,C 180,E1 -1328.225,E2 -1328.225} C_VEL
LIN {X 0,Y 587.348,Z 527.32,A -85,B 0,C 180,E1 -1331.151,E2 -1331.151} C_VEL
LIN {X 0,Y 587.326,Z 527.319,A -85,B 0,C 180,E1 -1334.024,E2 -1334.024} C_VEL
LIN {X 0,Y 587.361,Z 527.315,A -85,B 0,C 180,E1 -1336.154,E2 -1336.154} C_VEL
LIN {X 0,Y 587.341,Z 527.328,A -85,B 0,C 180,E1 -1338.962,E2 -1338.962} C_VEL
LIN {X 0,Y 587.368,Z 527.314,A -85,B 0,C 180,E1 -1341.744,E2 -1341.744} C_VEL
LIN {X 0,Y 587.357,Z 527.317,A -85,B 0,C 180,E1 -1344.507,E2 -1344.507} C_VEL
LIN {X 0,Y 587.373,Z 527.321,A -85,B 0,C 180,E1 -1347.256,E2 -1347.256} C_VEL
LIN {X 0,Y 587.383,Z 527.312,A -85,B 0,C 180,E1 -1350,E2 -1350} C_VEL
LIN {X 0,Y 587.369,Z 527.316,A -85,B 0,C 180,E1 -1352.743,E2 -1352.743} C_VEL
LIN {X 0,Y 587.367,Z 527.32,A -85,B 0,C 180,E1 -1355.492,E2 -1355.492} C_VEL
LIN {X 0,Y 587.364,Z 527.314,A -85,B 0,C 180,E1 -1358.255,E2 -1358.255} C_VEL
LIN {X 0,Y 587.345,Z 527.323,A -85,B 0,C 180,E1 -1361.133,E2 -1361.133} C_VEL
LIN {X 0,Y 587.363,Z 527.314,A -85,B 0,C 180,E1 -1364.26,E2 -1364.26} C_VEL
LIN {X 0,Y 587.357,Z 527.325,A -85,B 0,C 180,E1 -1367.405,E2 -1367.405} C_VEL
LIN {X 0,Y 587.329,Z 527.319,A -85,B 0,C 180,E1 -1370.304,E2 -1370.304} C_VEL
LIN {X 0,Y 587.32,Z 527.325,A -85,B 0,C 180,E1 -1373.258,E2 -1373.258} C_VEL
LIN {X 0,Y 587.336,Z 527.327,A -85,B 0,C 180,E1 -1375.516,E2 -1375.516} C_VEL
LIN {X 0,Y 587.346,Z 527.324,A -85,B 0,C 180,E1 -1377.817,E2 -1377.817} C_VEL
LIN {X 0,Y 587.346,Z 527.316,A -85,B 0,C 180,E1 -1380.512,E2 -1380.512} C_VEL
LIN {X 0,Y 587.334,Z 527.322,A -85,B 0,C 180,E1 -1383.396,E2 -1383.396} C_VEL
LIN {X 0,Y 587.353,Z 527.325,A -85,B 0,C 180,E1 -1385.895,E2 -1385.895} C_VEL
LIN {X 0,Y 587.329,Z 527.32,A -85,B 0,C 180,E1 -1388.479,E2 -1388.479} C_VEL
LIN {X 0,Y 587.335,Z 527.318,A -85,B 0,C 180,E1 -1391.156,E2 -1391.156} C_VEL
LIN {X 0,Y 587.322,Z 527.327,A -85,B 0,C 180,E1 -1394.113,E2 -1394.113} C_VEL
LIN {X 0,Y 587.318,Z 527.319,A -85,B 0,C 180,E1 -1396.994,E2 -1396.994} C_VEL
LIN {X 0,Y 587.317,Z 527.325,A -85,B 0,C 180,E1 -1399.746,E2 -1399.746} C_VEL
LIN {X 0,Y 587.344,Z 527.322,A -85,B 0,C 180,E1 -1402.393,E2 -1402.393} C_VEL
LIN {X 0,Y 587.343,Z 527.317,A -85,B 0,C 180,E1 -1404.946,E2 -1404.946} C_VEL
LIN {X 0,Y 587.335,Z 527.318,A -85,B 0,C 180,E1 -1407.421,E2 -1407.421} C_VEL
LIN {X 0,Y 587.344,Z 527.321,A -85,B 0,C 180,E1 -1409.831,E2 -1409.831} C_VEL
LIN {X 0,Y 587.321,Z 527.322,A -85,B 0,C 180,E1 -1411.623,E2 -1411.623} C_VEL
LIN {X 0,Y 588.071,Z 529.813,A -85,B 0,C 180,E1 -1411.685,E2 -1411.685} C_VEL
LIN {X 0,Y 588.011,Z 588.944,A -85,B 0,C 180,E1 -1412.434,E2 -1412.434} C_VEL
LIN {X 0,Y 587.907,Z 602.811,A -85,B 0,C 180,E1 -1412.742,E2 -1412.742} C_VEL
LIN {X 0,Y 587.818,Z 616.133,A -85,B 0,C 180,E1 -1413.171,E2 -1413.171} C_VEL
LIN {X 0,Y 587.745,Z 629.485,A -85,B 0,C 180,E1 -1413.741,E2 -1413.741} C_VEL
LIN {X 0,Y 587.639,Z 643.165,A -85,B 0,C 180,E1 -1414.498,E2 -1414.498} C_VEL
LIN {X 0,Y 587.532,Z 654.152,A -85,B 0,C 180,E1 -1415.25,E2 -1415.25} C_VEL
LIN {X 0,Y 587.433,Z 665.429,A -85,B 0,C 180,E1 -1416.186,E2 -1416.186} C_VEL
LIN {X 0,Y 587.348,Z 674.84,A -85,B 0,C 180,E1 -1417.123,E2 -1417.123} C_VEL
LIN {X 0,Y 587.306,Z 684.073,A -85,B 0,C 180,E1 -1418.225,E2 -1418.225} C_VEL
LIN {X 0,Y 587.245,Z 691.723,A -85,B 0,C 180,E1 -1419.334,E2 -1419.334} C_VEL
LIN {X 0,Y 587.227,Z 697.876,A -85,B 0,C 180,E1 -1420.421,E2 -1420.421} C_VEL
LIN {X 0,Y 587.2,Z 702.897,A -85,B 0,C 180,E1 -1421.509,E2 -1421.509} C_VEL
LIN {X 0,Y 587.155,Z 706.89,A -85,B 0,C 180,E1 -1422.588,E2 -1422.588} C_VEL
LIN {X 0,Y 587.159,Z 709.03,A -85,B 0,C 180,E1 -1423.306,E2 -1423.306} C_VEL
LIN {X 0,Y 587.141,Z 712.095,A -85,B 0,C 180,E1 -1424.732,E2 -1424.732} C_VEL
LIN {X 0,Y 587.156,Z 713.685,A -85,B 0,C 180,E1 -1426.15,E2 -1426.15} C_VEL
LIN {X 0,Y 587.156,Z 713.875,A -85,B 0,C 180,E1 -1427.558,E2 -1427.558} C_VEL
LIN {X 0,Y 587.157,Z 712.711,A -85,B 0,C 180,E1 -1428.959,E2 -1428.959} C_VEL
LIN {X 0,Y 587.149,Z 710.121,A -85,B 0,C 180,E1 -1430.353,E2 -1430.353} C_VEL
LIN {X 0,Y 587.186,Z 706.074,A -85,B 0,C 180,E1 -1431.743,E2 -1431.743} C_VEL
LIN {X 0,Y 587.208,Z 702.059,A -85,B 0,C 180,E1 -1432.781,E2 -1432.781} C_VEL
LIN {X 0,Y 587.203,Z 697.079,A -85,B 0,C 180,E1 -1433.817,E2 -1433.817} C_VEL
LIN {X 0,Y 587.274,Z 689.969,A -85,B 0,C 180,E1 -1435.023,E2 -1435.023} C_VEL
LIN {X 0,Y 587.297,Z 681.246,A -85,B 0,C 180,E1 -1436.227,E2 -1436.227} C_VEL
LIN {X 0,Y 587.384,Z 672.147,A -85,B 0,C 180,E1 -1437.257,E2 -1437.257} C_VEL
LIN {X 0,Y 587.464,Z 661.087,A -85,B 0,C 180,E1 -1438.286,E2 -1438.286} C_VEL
LIN {X 0,Y 587.573,Z 649.97,A -85,B 0,C 180,E1 -1439.144,E2 -1439.144} C_VEL
LIN {X 0,Y 587.674,Z 637.734,A -85,B 0,C 180,E1 -1439.915,E2 -1439.915} C_VEL
LIN {X 0,Y 587.785,Z 624.04,A -85,B 0,C 180,E1 -1440.6,E2 -1440.6} C_VEL
LIN {X 0,Y 587.872,Z 610.584,A -85,B 0,C 180,E1 -1441.113,E2 -1441.113} C_VEL
LIN {X 0,Y 587.959,Z 596.826,A -85,B 0,C 180,E1 -1441.499,E2 -1441.499} C_VEL
LIN {X 0,Y 588.011,Z 582.313,A -85,B 0,C 180,E1 -1441.755,E2 -1441.755} C_VEL
LIN {X 0,Y 588.001,Z 529.549,A -85,B 0,C 180,E1 -1442.41,E2 -1442.41} C_VEL
LIN {X 0,Y 587.364,Z 527.317,A -85,B 0,C 180,E1 -1442.465,E2 -1442.465} C_VEL
LIN {X 0,Y 587.351,Z 527.324,A -85,B 0,C 180,E1 -1445.493,E2 -1445.493} C_VEL
LIN {X 0,Y 587.368,Z 527.316,A -85,B 0,C 180,E1 -1448.256,E2 -1448.256} C_VEL
LIN {X 0,Y 587.345,Z 527.32,A -85,B 0,C 180,E1 -1451.134,E2 -1451.134} C_VEL
LIN {X 0,Y 587.362,Z 527.317,A -85,B 0,C 180,E1 -1454.261,E2 -1454.261} C_VEL
LIN {X 0,Y 587.347,Z 527.325,A -85,B 0,C 180,E1 -1457.406,E2 -1457.406} C_VEL
LIN {X 0,Y 587.328,Z 527.32,A -85,B 0,C 180,E1 -1460.305,E2 -1460.305} C_VEL
LIN {X 0,Y 587.322,Z 527.327,A -85,B 0,C 180,E1 -1463.259,E2 -1463.259} C_VEL
LIN {X 0,Y 587.336,Z 527.327,A -85,B 0,C 180,E1 -1465.517,E2 -1465.517} C_VEL
LIN {X 0,Y 587.346,Z 527.32,A -85,B 0,C 180,E1 -1467.818,E2 -1467.818} C_VEL
LIN {X 0,Y 587.35,Z 527.316,A -85,B 0,C 180,E1 -1470.513,E2 -1470.513} C_VEL
LIN {X 0,Y 587.335,Z 527.327,A -85,B 0,C 180,E1 -1473.397,E2 -1473.397} C_VEL
LIN {X 0,Y 587.296,Z 527.324,A -85,B 0,C 180,E1 -1475.9,E2 -1475.9} C_VEL
LIN {X 0,Y 587.333,Z 527.319,A -85,B 0,C 180,E1 -1478.479,E2 -1478.479} C_VEL
LIN {X 0,Y 587.336,Z 527.327,A -85,B 0,C 180,E1 -1481.157,E2 -1481.157} C_VEL
LIN {X 0,Y 587.334,Z 527.318,A -85,B 0,C 180,E1 -1484.115,E2 -1484.115} C_VEL
LIN {X 0,Y 587.312,Z 527.328,A -85,B 0,C 180,E1 -1486.994,E2 -1486.994} C_VEL
LIN {X 0,Y 587.318,Z 527.322,A -85,B 0,C 180,E1 -1489.747,E2 -1489.747} C_VEL
LIN {X 0,Y 587.345,Z 527.318,A -85,B 0,C 180,E1 -1492.393,E2 -1492.393} C_VEL
LIN {X 0,Y 587.351,Z 527.325,A -85,B 0,C 180,E1 -1494.947,E2 -1494.947} C_VEL
LIN {X 0,Y 587.342,Z 527.324,A -85,B 0,C 180,E1 -1497.422,E2 -1497.422} C_VEL
LIN {X 0,Y 587.395,Z 527.491,A -85,B 0,C 180,E1 -1499.361,E2 -1499.361} C_VEL
LIN {X 0,Y 588.357,Z 532.377,A -85,B 0,C 180,E1 -1500.086,E2 -1500.086} C_VEL
LIN {X 0,Y 588.243,Z 548.654,A -85,B 0,C 180,E1 -1502.422,E2 -1502.422} C_VEL
LIN {X 0,Y 588.064,Z 567.367,A -85,B 0,C 180,E1 -1505.085,E2 -1505.085} C_VEL
LIN {X 0,Y 587.873,Z 588.753,A -85,B 0,C 180,E1 -1508.063,E2 -1508.063} C_VEL
LIN {X 0,Y 587.694,Z 609.256,A -85,B 0,C 180,E1 -1510.862,E2 -1510.862} C_VEL
LIN {X 0,Y 587.552,Z 630.189,A -85,B 0,C 180,E1 -1513.675,E2 -1513.675} C_VEL
LIN {X 0,Y 587.412,Z 651.491,A -85,B 0,C 180,E1 -1516.498,E2 -1516.498} C_VEL
LIN {X 0,Y 587.903,Z 655.757,A -85,B 0,C 180,E1 -1516.564,E2 -1516.564} C_VEL
LIN {X 0,Y 587.72,Z 759.969,A -85,B 0,C 180,E1 -1517.855,E2 -1517.855} C_VEL
LIN {X 0,Y 587.675,Z 773.232,A -85,B 0,C 180,E1 -1518.161,E2 -1518.161} C_VEL
LIN {X 0,Y 587.638,Z 785.773,A -85,B 0,C 180,E1 -1518.591,E2 -1518.591} C_VEL
LIN {X 0,Y 587.553,Z 797.64,A -85,B 0,C 180,E1 -1519.141,E2 -1519.141} C_VEL
LIN {X 0,Y 587.462,Z 809.206,A -85,B 0,C 180,E1 -1519.837,E2 -1519.837} C_VEL
LIN {X 0,Y 587.391,Z 819.601,A -85,B 0,C 180,E1 -1520.618,E2 -1520.618} C_VEL
LIN {X 0,Y 587.321,Z 828.117,A -85,B 0,C 180,E1 -1521.398,E2 -1521.398} C_VEL
LIN {X 0,Y 587.273,Z 835.964,A -85,B 0,C 180,E1 -1522.263,E2 -1522.263} C_VEL
LIN {X 0,Y 587.23,Z 842.473,A -85,B 0,C 180,E1 -1523.127,E2 -1523.127} C_VEL
LIN {X 0,Y 587.236,Z 848.869,A -85,B 0,C 180,E1 -1524.162,E2 -1524.162} C_VEL
LIN {X 0,Y 587.147,Z 853.951,A -85,B 0,C 180,E1 -1525.194,E2 -1525.194} C_VEL
LIN {X 0,Y 587.213,Z 857.897,A -85,B 0,C 180,E1 -1526.226,E2 -1526.226} C_VEL
LIN {X 0,Y 587.132,Z 860.811,A -85,B 0,C 180,E1 -1527.256,E2 -1527.256} C_VEL
LIN {X 0,Y 587.138,Z 862.202,A -85,B 0,C 180,E1 -1527.942,E2 -1527.942} C_VEL
LIN {X 0,Y 587.14,Z 863.785,A -85,B 0,C 180,E1 -1529.315,E2 -1529.315} C_VEL
LIN {X 0,Y 587.137,Z 864,A -85,B 0,C 180,E1 -1530,E2 -1530} C_VEL
LIN {X 0,Y 587.147,Z 863.184,A -85,B 0,C 180,E1 -1531.372,E2 -1531.372} C_VEL
LIN {X 0,Y 587.138,Z 862.2,A -85,B 0,C 180,E1 -1532.058,E2 -1532.058} C_VEL
LIN {X 0,Y 587.132,Z 860.808,A -85,B 0,C 180,E1 -1532.745,E2 -1532.745} C_VEL
LIN {X 0,Y 587.213,Z 857.895,A -85,B 0,C 180,E1 -1533.775,E2 -1533.775} C_VEL
LIN {X 0,Y 587.147,Z 853.948,A -85,B 0,C 180,E1 -1534.807,E2 -1534.807} C_VEL
LIN {X 0,Y 587.217,Z 847.875,A -85,B 0,C 180,E1 -1536.012,E2 -1536.012} C_VEL
LIN {X 0,Y 587.245,Z 841.234,A -85,B 0,C 180,E1 -1537.047,E2 -1537.047} C_VEL
LIN {X 0,Y 587.3,Z 832.987,A -85,B 0,C 180,E1 -1538.083,E2 -1538.083} C_VEL
LIN {X 0,Y 587.344,Z 824.533,A -85,B 0,C 180,E1 -1538.949,E2 -1538.949} C_VEL
LIN {X 0,Y 587.412,Z 814.089,A -85,B 0,C 180,E1 -1539.817,E2 -1539.817} C_VEL
LIN {X 0,Y 587.507,Z 803.752,A -85,B 0,C 180,E1 -1540.512,E2 -1540.512} C_VEL
LIN {X 0,Y 587.584,Z 791.797,A -85,B 0,C 180,E1 -1541.149,E2 -1541.149} C_VEL
LIN {X 0,Y 587.629,Z 779.586,A -85,B 0,C 180,E1 -1541.64,E2 -1541.64} C_VEL
LIN {X 0,Y 587.7,Z 766.425,A -85,B 0,C 180,E1 -1542.014,E2 -1542.014} C_VEL
LIN {X 0,Y 587.769,Z 754.056,A -85,B 0,C 180,E1 -1542.232,E2 -1542.232} C_VEL
LIN {X 0,Y 587.737,Z 653.453,A -85,B 0,C 180,E1 -1543.468,E2 -1543.468} C_VEL
LIN {X 0,Y 587.415,Z 651.401,A -85,B 0,C 180,E1 -1543.514,E2 -1543.514} C_VEL
LIN {X 0,Y 587.567,Z 628.846,A -85,B 0,C 180,E1 -1546.504,E2 -1546.504} C_VEL
LIN {X 0,Y 587.738,Z 607.133,A -85,B 0,C 180,E1 -1549.424,E2 -1549.424} C_VEL
LIN {X 0,Y 587.902,Z 584.737,A -85,B 0,C 180,E1 -1552.491,E2 -1552.491} C_VEL
LIN {X 0,Y 588.091,Z 563.351,A -85,B 0,C 180,E1 -1555.482,E2 -1555.482} C_VEL
LIN {X 0,Y 588.296,Z 544.641,A -85,B 0,C 180,E1 -1558.156,E2 -1558.156} C_VEL
LIN {X 0,Y 588.337,Z 532.246,A -85,B 0,C 180,E1 -1559.916,E2 -1559.916} C_VEL
LIN {X 0,Y 587.362,Z 527.322,A -85,B 0,C 180,E1 -1560.577,E2 -1560.577} C_VEL
LIN {X 0,Y 587.339,Z 527.322,A -85,B 0,C 180,E1 -1563.397,E2 -1563.397} C_VEL
LIN {X 0,Y 587.298,Z 527.323,A -85,B 0,C 180,E1 -1565.9,E2 -1565.9} C_VEL
LIN {X 0,Y 587.335,Z 527.322,A -85,B 0,C 180,E1 -1568.479,E2 -1568.479} C_VEL
LIN {X 0,Y 587.339,Z 527.323,A -85,B 0,C 180,E1 -1571.157,E2 -1571.157} C_VEL
LIN {X 0,Y 587.316,Z 527.322,A -85,B 0,C 180,E1 -1574.112,E2 -1574.112} C_VEL
LIN {X 0,Y 587.319,Z 527.326,A -85,B 0,C 180,E1 -1576.994,E2 -1576.994} C_VEL
LIN {X 0,Y 587.321,Z 527.32,A -85,B 0,C 180,E1 -1579.746,E2 -1579.746} C_VEL
LIN {X 0,Y 587.35,Z 527.322,A -85,B 0,C 180,E1 -1582.392,E2 -1582.392} C_VEL
LIN {X 0,Y 587.364,Z 527.315,A -85,B 0,C 180,E1 -1585.78,E2 -1585.78} C_VEL
LIN {X 0,Y 587.354,Z 527.321,A -85,B 0,C 180,E1 -1588.232,E2 -1588.232} C_VEL
LIN {X 0,Y 587.354,Z 527.321,A -85,B 0,C 180,E1 -1590.866,E2 -1590.866} C_VEL
LIN {X 0,Y 587.364,Z 527.316,A -85,B 0,C 180,E1 -1593.819,E2 -1593.819} C_VEL
LIN {X 0,Y 587.339,Z 527.321,A -85,B 0,C 180,E1 -1595.993,E2 -1595.993} C_VEL
LIN {X 0,Y 587.335,Z 527.321,A -85,B 0,C 180,E1 -1598.962,E2 -1598.962} C_VEL
LIN {X 0,Y 587.351,Z 527.318,A -85,B 0,C 180,E1 -1601.151,E2 -1601.151} C_VEL
LIN {X 0,Y 587.322,Z 527.326,A -85,B 0,C 180,E1 -1604.024,E2 -1604.024} C_VEL
LIN {X 0,Y 587.337,Z 527.32,A -85,B 0,C 180,E1 -1605.472,E2 -1605.472} C_VEL
LIN {X 0,Y 588.359,Z 530.715,A -85,B 0,C 180,E1 -1605.548,E2 -1605.548} C_VEL
LIN {X 0,Y 588.277,Z 569.174,A -85,B 0,C 180,E1 -1606.053,E2 -1606.053} C_VEL
LIN {X 0,Y 588.199,Z 584.709,A -85,B 0,C 180,E1 -1606.394,E2 -1606.394} C_VEL
LIN {X 0,Y 588.074,Z 599.651,A -85,B 0,C 180,E1 -1606.875,E2 -1606.875} C_VEL
LIN {X 0,Y 587.982,Z 614.205,A -85,B 0,C 180,E1 -1607.488,E2 -1607.488} C_VEL
LIN {X 0,Y 587.877,Z 627.359,A -85,B 0,C 180,E1 -1608.186,E2 -1608.186} C_VEL
LIN {X 0,Y 587.699,Z 640.811,A -85,B 0,C 180,E1 -1609.056,E2 -1609.056} C_VEL
LIN {X 0,Y 587.587,Z 653.033,A -85,B 0,C 180,E1 -1610.012,E2 -1610.012} C_VEL
LIN {X 0,Y 587.47,Z 664.182,A -85,B 0,C 180,E1 -1611.053,E2 -1611.053} C_VEL
LIN {X 0,Y 587.371,Z 675.054,A -85,B 0,C 180,E1 -1612.264,E2 -1612.264} C_VEL
LIN {X 0,Y 587.326,Z 684.644,A -85,B 0,C 180,E1 -1613.552,E2 -1613.552} C_VEL
LIN {X 0,Y 587.259,Z 692.602,A -85,B 0,C 180,E1 -1614.85,E2 -1614.85} C_VEL
LIN {X 0,Y 587.211,Z 699.452,A -85,B 0,C 180,E1 -1616.225,E2 -1616.225} C_VEL
LIN {X 0,Y 587.17,Z 704.846,A -85,B 0,C 180,E1 -1617.599,E2 -1617.599} C_VEL
LIN {X 0,Y 587.155,Z 708.028,A -85,B 0,C 180,E1 -1618.628,E2 -1618.628} C_VEL
LIN {X 0,Y 587.133,Z 711.187,A -85,B 0,C 180,E1 -1620,E2 -1620} C_VEL
LIN {X 0,Y 587.143,Z 713.139,A -85,B 0,C 180,E1 -1621.371,E2 -1621.371} C_VEL
LIN {X 0,Y 587.128,Z 713.944,A -85,B 0,C 180,E1 -1622.744,E2 -1622.744} C_VEL
LIN {X 0,Y 587.165,Z 713.624,A -85,B 0,C 180,E1 -1624.118,E2 -1624.118} C_VEL
LIN {X 0,Y 587.163,Z 712.17,A -85,B 0,C 180,E1 -1625.494,E2 -1625.494} C_VEL
LIN {X 0,Y 587.166,Z 709.536,A -85,B 0,C 180,E1 -1626.874,E2 -1626.874} C_VEL
LIN {X 0,Y 587.188,Z 705.637,A -85,B 0,C 180,E1 -1628.257,E2 -1628.257} C_VEL
LIN {X 0,Y 587.196,Z 700.401,A -85,B 0,C 180,E1 -1629.646,E2 -1629.646} C_VEL
LIN {X 0,Y 587.246,Z 693.46,A -85,B 0,C 180,E1 -1631.081,E2 -1631.081} C_VEL
LIN {X 0,Y 587.282,Z 685.297,A -85,B 0,C 180,E1 -1632.439,E2 -1632.439} C_VEL
LIN {X 0,Y 587.357,Z 676.318,A -85,B 0,C 180,E1 -1633.669,E2 -1633.669} C_VEL
LIN {X 0,Y 587.464,Z 665.477,A -85,B 0,C 180,E1 -1634.904,E2 -1634.904} C_VEL
LIN {X 0,Y 587.575,Z 654.31,A -85,B 0,C 180,E1 -1635.968,E2 -1635.968} C_VEL
LIN {X 0,Y 587.624,Z 647.84,A -85,B 0,C 180,E1 -1636.505,E2 -1636.505} C_VEL
LIN {X 0,Y 586.991,Z 643.323,A -85,B 0,C 180,E1 -1636.867,E2 -1636.867} C_VEL
LIN {X 0,Y 581.977,Z 629.858,A -85,B 0,C 180,E1 -1637.906,E2 -1637.906} C_VEL
LIN {X 0,Y 581.025,Z 624.974,A -85,B 0,C 180,E1 -1638.221,E2 -1638.221} C_VEL
LIN {X 0,Y 580.964,Z 623.255,A -85,B 0,C 180,E1 -1638.32,E2 -1638.32} C_VEL
LIN {X 0,Y 581.187,Z 608.429,A -85,B 0,C 180,E1 -1639.056,E2 -1639.056} C_VEL
LIN {X 0,Y 581.318,Z 594.118,A -85,B 0,C 180,E1 -1639.607,E2 -1639.607} C_VEL
LIN {X 0,Y 581.447,Z 579.238,A -85,B 0,C 180,E1 -1640.035,E2 -1640.035} C_VEL
LIN {X 0,Y 581.524,Z 563.549,A -85,B 0,C 180,E1 -1640.332,E2 -1640.332} C_VEL
LIN {X 0,Y 581.516,Z 531.954,A -85,B 0,C 180,E1 -1640.738,E2 -1640.738} C_VEL
LIN {X 0,Y 580.309,Z 528.195,A -85,B 0,C 180,E1 -1640.834,E2 -1640.834} C_VEL
LIN {X 0,Y 580.275,Z 528.203,A -85,B 0,C 180,E1 -1643.558,E2 -1643.558} C_VEL
LIN {X 0,Y 580.292,Z 528.204,A -85,B 0,C 180,E1 -1645.849,E2 -1645.849} C_VEL
LIN {X 0,Y 580.302,Z 528.202,A -85,B 0,C 180,E1 -1648.185,E2 -1648.185} C_VEL
LIN {X 0,Y 580.285,Z 528.197,A -85,B 0,C 180,E1 -1650.694,E2 -1650.694} C_VEL
LIN {X 0,Y 580.303,Z 528.194,A -85,B 0,C 180,E1 -1653.316,E2 -1653.316} C_VEL
LIN {X 0,Y 580.246,Z 528.205,A -85,B 0,C 180,E1 -1655.756,E2 -1655.756} C_VEL
LIN {X 0,Y 580.291,Z 528.205,A -85,B 0,C 180,E1 -1658.146,E2 -1658.146} C_VEL
LIN {X 0,Y 580.3,Z 528.195,A -85,B 0,C 180,E1 -1660.843,E2 -1660.843} C_VEL
LIN {X 0,Y 580.289,Z 528.197,A -85,B 0,C 180,E1 -1663.656,E2 -1663.656} C_VEL
LIN {X 0,Y 580.273,Z 528.203,A -85,B 0,C 180,E1 -1666.609,E2 -1666.609} C_VEL
LIN {X 0,Y 580.298,Z 528.195,A -85,B 0,C 180,E1 -1669.156,E2 -1669.156} C_VEL
LIN {X 0,Y 580.289,Z 528.198,A -85,B 0,C 180,E1 -1671.927,E2 -1671.927} C_VEL
LIN {X 0,Y 580.281,Z 528.207,A -85,B 0,C 180,E1 -1674.454,E2 -1674.454} C_VEL
LIN {X 0,Y 580.292,Z 528.198,A -85,B 0,C 180,E1 -1676.975,E2 -1676.975} C_VEL
LIN {X 0,Y 580.298,Z 528.194,A -85,B 0,C 180,E1 -1679.425,E2 -1679.425} C_VEL
LIN {X 0,Y 580.297,Z 528.197,A -85,B 0,C 180,E1 -1682.141,E2 -1682.141} C_VEL
LIN {X 0,Y 580.321,Z 528.193,A -85,B 0,C 180,E1 -1685.269,E2 -1685.269} C_VEL
LIN {X 0,Y 580.273,Z 528.197,A -85,B 0,C 180,E1 -1687.947,E2 -1687.947} C_VEL
LIN {X 0,Y 580.318,Z 528.2,A -85,B 0,C 180,E1 -1690.914,E2 -1690.914} C_VEL
LIN {X 0,Y 580.28,Z 528.196,A -85,B 0,C 180,E1 -1693.825,E2 -1693.825} C_VEL
LIN {X 0,Y 580.326,Z 528.19,A -85,B 0,C 180,E1 -1695.983,E2 -1695.983} C_VEL
LIN {X 0,Y 580.304,Z 528.202,A -85,B 0,C 180,E1 -1698.826,E2 -1698.826} C_VEL
LIN {X 0,Y 580.332,Z 528.191,A -85,B 0,C 180,E1 -1701.644,E2 -1701.644} C_VEL
LIN {X 0,Y 580.323,Z 528.193,A -85,B 0,C 180,E1 -1704.44,E2 -1704.44} C_VEL
LIN {X 0,Y 580.339,Z 528.197,A -85,B 0,C 180,E1 -1707.223,E2 -1707.223} C_VEL
LIN {X 0,Y 580.352,Z 528.187,A -85,B 0,C 180,E1 -1710,E2 -1710} C_VEL
LIN {X 0,Y 580.336,Z 528.193,A -85,B 0,C 180,E1 -1712.776,E2 -1712.776} C_VEL
LIN {X 0,Y 580.332,Z 528.195,A -85,B 0,C 180,E1 -1715.559,E2 -1715.559} C_VEL
LIN {X 0,Y 580.327,Z 528.19,A -85,B 0,C 180,E1 -1718.356,E2 -1718.356} C_VEL
LIN {X 0,Y 580.297,Z 528.202,A -85,B 0,C 180,E1 -1721.191,E2 -1721.191} C_VEL
LIN {X 0,Y 580.325,Z 528.192,A -85,B 0,C 180,E1 -1724.016,E2 -1724.016} C_VEL
LIN {X 0,Y 580.309,Z 528.195,A -85,B 0,C 180,E1 -1726.914,E2 -1726.914} C_VEL
LIN {X 0,Y 580.304,Z 528.199,A -85,B 0,C 180,E1 -1729.822,E2 -1729.822} C_VEL
LIN {X 0,Y 580.292,Z 528.195,A -85,B 0,C 180,E1 -1732.802,E2 -1732.802} C_VEL
LIN {X 0,Y 580.306,Z 528.195,A -85,B 0,C 180,E1 -1735.079,E2 -1735.079} C_VEL
LIN {X 0,Y 580.317,Z 528.199,A -85,B 0,C 180,E1 -1737.863,E2 -1737.863} C_VEL
LIN {X 0,Y 580.294,Z 528.194,A -85,B 0,C 180,E1 -1740.697,E2 -1740.697} C_VEL
LIN {X 0,Y 580.302,Z 528.197,A -85,B 0,C 180,E1 -1743.317,E2 -1743.317} C_VEL
LIN {X 0,Y 580.323,Z 528.201,A -85,B 0,C 180,E1 -1745.767,E2 -1745.767} C_VEL
LIN {X 0,Y 580.285,Z 528.201,A -85,B 0,C 180,E1 -1748.146,E2 -1748.146} C_VEL
LIN {X 0,Y 580.3,Z 528.194,A -85,B 0,C 180,E1 -1750.843,E2 -1750.843} C_VEL
LIN {X 0,Y 580.274,Z 528.203,A -85,B 0,C 180,E1 -1753.658,E2 -1753.658} C_VEL
LIN {X 0,Y 580.281,Z 528.198,A -85,B 0,C 180,E1 -1756.608,E2 -1756.608} C_VEL
LIN {X 0,Y 580.297,Z 528.194,A -85,B 0,C 180,E1 -1759.157,E2 -1759.157} C_VEL
LIN {X 0,Y 580.288,Z 528.203,A -85,B 0,C 180,E1 -1761.926,E2 -1761.926} C_VEL
LIN {X 0,Y 580.301,Z 528.199,A -85,B 0,C 180,E1 -1764.457,E2 -1764.457} C_VEL
LIN {X 0,Y 580.287,Z 528.196,A -85,B 0,C 180,E1 -1766.975,E2 -1766.975} C_VEL
LIN {X 0,Y 580.306,Z 528.195,A -85,B 0,C 180,E1 -1769.426,E2 -1769.426} C_VEL
LIN {X 0,Y 580.286,Z 528.231,A -85,B 0,C 180,E1 -1771.454,E2 -1771.454} C_VEL
LIN {X 0,Y 581.267,Z 531.901,A -85,B 0,C 180,E1 -1771.527,E2 -1771.527} C_VEL
LIN {X 0,Y 581.138,Z 589.478,A -85,B 0,C 180,E1 -1772.268,E2 -1772.268} C_VEL
LIN {X 0,Y 581.006,Z 603.557,A -85,B 0,C 180,E1 -1772.591,E2 -1772.591} C_VEL
LIN {X 0,Y 580.952,Z 615.328,A -85,B 0,C 180,E1 -1772.974,E2 -1772.974} C_VEL
LIN {X 0,Y 580.834,Z 627.409,A -85,B 0,C 180,E1 -1773.483,E2 -1773.483} C_VEL
LIN {X 0,Y 580.663,Z 638.834,A -85,B 0,C 180,E1 -1774.084,E2 -1774.084} C_VEL
LIN {X 0,Y 580.588,Z 650.523,A -85,B 0,C 180,E1 -1774.838,E2 -1774.838} C_VEL
LIN {X 0,Y 580.459,Z 662.501,A -85,B 0,C 180,E1 -1775.786,E2 -1775.786} C_VEL
LIN {X 0,Y 580.331,Z 672.553,A -85,B 0,C 180,E1 -1776.756,E2 -1776.756} C_VEL
LIN {X 0,Y 580.253,Z 681.281,A -85,B 0,C 180,E1 -1777.76,E2 -1777.76} C_VEL
LIN {X 0,Y 580.22,Z 689.236,A -85,B 0,C 180,E1 -1778.854,E2 -1778.854} C_VEL
LIN {X 0,Y 580.141,Z 697.008,A -85,B 0,C 180,E1 -1780.172,E2 -1780.172} C_VEL
LIN {X 0,Y 580.106,Z 702.22,A -85,B 0,C 180,E1 -1781.274,E2 -1781.274} C_VEL
LIN {X 0,Y 580.073,Z 706.375,A -85,B 0,C 180,E1 -1782.369,E2 -1782.369} C_VEL
LIN {X 0,Y 580.045,Z 708.802,A -85,B 0,C 180,E1 -1783.172,E2 -1783.172} C_VEL
LIN {X 0,Y 580.058,Z 711.838,A -85,B 0,C 180,E1 -1784.541,E2 -1784.541} C_VEL
LIN {X 0,Y 580.069,Z 713.574,A -85,B 0,C 180,E1 -1785.977,E2 -1785.977} C_VEL
LIN {X 0,Y 580.054,Z 713.937,A -85,B 0,C 180,E1 -1786.691,E2 -1786.691} C_VEL
LIN {X 0,Y 580.048,Z 713.591,A -85,B 0,C 180,E1 -1788.114,E2 -1788.114} C_VEL
LIN {X 0,Y 580.055,Z 711.855,A -85,B 0,C 180,E1 -1789.529,E2 -1789.529} C_VEL
LIN {X 0,Y 580.055,Z 710.492,A -85,B 0,C 180,E1 -1790.234,E2 -1790.234} C_VEL
LIN {X 0,Y 580.107,Z 706.615,A -85,B 0,C 180,E1 -1791.641,E2 -1791.641} C_VEL
LIN {X 0,Y 580.117,Z 702.725,A -85,B 0,C 180,E1 -1792.692,E2 -1792.692} C_VEL
LIN {X 0,Y 580.103,Z 697.903,A -85,B 0,C 180,E1 -1793.741,E2 -1793.741} C_VEL
LIN {X 0,Y 580.189,Z 690.976,A -85,B 0,C 180,E1 -1794.962,E2 -1794.962} C_VEL
LIN {X 0,Y 580.218,Z 683.795,A -85,B 0,C 180,E1 -1796.007,E2 -1796.007} C_VEL
LIN {X 0,Y 580.305,Z 675.22,A -85,B 0,C 180,E1 -1797.05,E2 -1797.05} C_VEL
LIN {X 0,Y 580.431,Z 664.865,A -85,B 0,C 180,E1 -1798.092,E2 -1798.092} C_VEL
LIN {X 0,Y 580.528,Z 653.339,A -85,B 0,C 180,E1 -1799.047,E2 -1799.047} C_VEL
LIN {X 0,Y 580.646,Z 641.812,A -85,B 0,C 180,E1 -1799.827,E2 -1799.827} C_VEL
LIN {X 0,Y 580.803,Z 630.935,A -85,B 0,C 180,E1 -1800.434,E2 -1800.434} C_VEL
LIN {X 0,Y 580.942,Z 617.393,A -85,B 0,C 180,E1 -1801.04,E2 -1801.04} C_VEL
LIN {X 0,Y 581.037,Z 602.231,A -85,B 0,C 180,E1 -1801.538,E2 -1801.538} C_VEL
LIN {X 0,Y 581.135,Z 588.446,A -85,B 0,C 180,E1 -1801.841,E2 -1801.841} C_VEL
LIN {X 0,Y 581.139,Z 530.968,A -85,B 0,C 180,E1 -1802.578,E2 -1802.578} C_VEL
LIN {X 0,Y 580.343,Z 528.191,A -85,B 0,C 180,E1 -1802.647,E2 -1802.647} C_VEL
LIN {X 0,Y 580.317,Z 528.201,A -85,B 0,C 180,E1 -1805.56,E2 -1805.56} C_VEL
LIN {X 0,Y 580.331,Z 528.192,A -85,B 0,C 180,E1 -1808.356,E2 -1808.356} C_VEL
LIN {X 0,Y 580.296,Z 528.199,A -85,B 0,C 180,E1 -1811.191,E2 -1811.191} C_VEL
LIN {X 0,Y 580.323,Z 528.196,A -85,B 0,C 180,E1 -1814.017,E2 -1814.017} C_VEL
LIN {X 0,Y 580.309,Z 528.195,A -85,B 0,C 180,E1 -1816.914,E2 -1816.914} C_VEL
LIN {X 0,Y 580.303,Z 528.2,A -85,B 0,C 180,E1 -1819.823,E2 -1819.823} C_VEL
LIN {X 0,Y 580.294,Z 528.197,A -85,B 0,C 180,E1 -1822.803,E2 -1822.803} C_VEL
LIN {X 0,Y 580.307,Z 528.198,A -85,B 0,C 180,E1 -1825.08,E2 -1825.08} C_VEL
LIN {X 0,Y 580.297,Z 528.198,A -85,B 0,C 180,E1 -1827.86,E2 -1827.86} C_VEL
LIN {X 0,Y 580.298,Z 528.195,A -85,B 0,C 180,E1 -1830.698,E2 -1830.698} C_VEL
LIN {X 0,Y 580.303,Z 528.203,A -85,B 0,C 180,E1 -1833.317,E2 -1833.317} C_VEL
LIN {X 0,Y 580.259,Z 528.202,A -85,B 0,C 180,E1 -1835.759,E2 -1835.759} C_VEL
LIN {X 0,Y 580.289,Z 528.196,A -85,B 0,C 180,E1 -1838.147,E2 -1838.147} C_VEL
LIN {X 0,Y 580.299,Z 528.199,A -85,B 0,C 180,E1 -1840.844,E2 -1840.844} C_VEL
LIN {X 0,Y 580.287,Z 528.199,A -85,B 0,C 180,E1 -1843.657,E2 -1843.657} C_VEL
LIN {X 0,Y 580.275,Z 528.2,A -85,B 0,C 180,E1 -1846.61,E2 -1846.61} C_VEL
LIN {X 0,Y 580.299,Z 528.204,A -85,B 0,C 180,E1 -1849.157,E2 -1849.157} C_VEL
LIN {X 0,Y 580.29,Z 528.197,A -85,B 0,C 180,E1 -1851.928,E2 -1851.928} C_VEL
LIN {X 0,Y 580.3,Z 528.197,A -85,B 0,C 180,E1 -1854.457,E2 -1854.457} C_VEL
LIN {X 0,Y 580.293,Z 528.206,A -85,B 0,C 180,E1 -1856.976,E2 -1856.976} C_VEL
LIN {X 0,Y 580.311,Z 528.224,A -85,B 0,C 180,E1 -1859.132,E2 -1859.132} C_VEL
LIN {X 0,Y 581.501,Z 534.578,A -85,B 0,C 180,E1 -1860.097,E2 -1860.097} C_VEL
LIN {X 0,Y 581.443,Z 551.38,A -85,B 0,C 180,E1 -1862.47,E2 -1862.47} C_VEL
LIN {X 0,Y 581.174,Z 570.404,A -85,B 0,C 180,E1 -1865.204,E2 -1865.204} C_VEL
LIN {X 0,Y 580.975,Z 590.09,A -85,B 0,C 180,E1 -1867.976,E2 -1867.976} C_VEL
LIN {X 0,Y 580.749,Z 609.968,A -85,B 0,C 180,E1 -1870.722,E2 -1870.722} C_VEL
LIN {X 0,Y 580.583,Z 630.189,A -85,B 0,C 180,E1 -1873.473,E2 -1873.473} C_VEL
LIN {X 0,Y 580.405,Z 651.491,A -85,B 0,C 180,E1 -1876.332,E2 -1876.332} C_VEL
LIN {X 0,Y 580.985,Z 655.757,A -85,B 0,C 180,E1 -1876.401,E2 -1876.401} C_VEL
LIN {X 0,Y 580.802,Z 759.969,A -85,B 0,C 180,E1 -1877.709,E2 -1877.709} C_VEL
LIN {X 0,Y 580.746,Z 773.232,A -85,B 0,C 180,E1 -1878.018,E2 -1878.018} C_VEL
LIN {X 0,Y 580.668,Z 785.382,A -85,B 0,C 180,E1 -1878.437,E2 -1878.437} C_VEL
LIN {X 0,Y 580.563,Z 797.639,A -85,B 0,C 180,E1 -1879.009,E2 -1879.009} C_VEL
LIN {X 0,Y 580.431,Z 809.207,A -85,B 0,C 180,E1 -1879.712,E2 -1879.712} C_VEL
LIN {X 0,Y 580.341,Z 819.602,A -85,B 0,C 180,E1 -1880.503,E2 -1880.503} C_VEL
LIN {X 0,Y 580.271,Z 828.117,A -85,B 0,C 180,E1 -1881.293,E2 -1881.293} C_VEL
LIN {X 0,Y 580.221,Z 835.964,A -85,B 0,C 180,E1 -1882.169,E2 -1882.169} C_VEL
LIN {X 0,Y 580.153,Z 843.652,A -85,B 0,C 180,E1 -1883.222,E2 -1883.222} C_VEL
LIN {X 0,Y 580.139,Z 850.683,A -85,B 0,C 180,E1 -1884.439,E2 -1884.439} C_VEL
LIN {X 0,Y 580.108,Z 855.372,A -85,B 0,C 180,E1 -1885.484,E2 -1885.484} C_VEL
LIN {X 0,Y 580.123,Z 858.958,A -85,B 0,C 180,E1 -1886.528,E2 -1886.528} C_VEL
LIN {X 0,Y 580.043,Z 860.811,A -85,B 0,C 180,E1 -1887.222,E2 -1887.222} C_VEL
LIN {X 0,Y 580.038,Z 862.202,A -85,B 0,C 180,E1 -1887.917,E2 -1887.917} C_VEL
LIN {X 0,Y 580.04,Z 863.785,A -85,B 0,C 180,E1 -1889.306,E2 -1889.306} C_VEL
LIN {X 0,Y 580.037,Z 864,A -85,B 0,C 180,E1 -1890,E2 -1890} C_VEL
LIN {X 0,Y 580.047,Z 863.185,A -85,B 0,C 180,E1 -1891.389,E2 -1891.389} C_VEL
LIN {X 0,Y 580.038,Z 862.2,A -85,B 0,C 180,E1 -1892.084,E2 -1892.084} C_VEL
LIN {X 0,Y 580.043,Z 860.808,A -85,B 0,C 180,E1 -1892.778,E2 -1892.778} C_VEL
LIN {X 0,Y 580.11,Z 857.895,A -85,B 0,C 180,E1 -1893.821,E2 -1893.821} C_VEL
LIN {X 0,Y 580.054,Z 853.948,A -85,B 0,C 180,E1 -1894.866,E2 -1894.866} C_VEL
LIN {X 0,Y 580.139,Z 847.874,A -85,B 0,C 180,E1 -1896.085,E2 -1896.085} C_VEL
LIN {X 0,Y 580.185,Z 841.234,A -85,B 0,C 180,E1 -1897.133,E2 -1897.133} C_VEL
LIN {X 0,Y 580.251,Z 832.987,A -85,B 0,C 180,E1 -1898.182,E2 -1898.182} C_VEL
LIN {X 0,Y 580.308,Z 824.533,A -85,B 0,C 180,E1 -1899.059,E2 -1899.059} C_VEL
LIN {X 0,Y 580.417,Z 814.091,A -85,B 0,C 180,E1 -1899.936,E2 -1899.936} C_VEL
LIN {X 0,Y 580.513,Z 803.751,A -85,B 0,C 180,E1 -1900.64,E2 -1900.64} C_VEL
LIN {X 0,Y 580.598,Z 792.229,A -85,B 0,C 180,E1 -1901.265,E2 -1901.265} C_VEL
LIN {X 0,Y 580.671,Z 779.465,A -85,B 0,C 180,E1 -1901.785,E2 -1901.785} C_VEL
LIN {X 0,Y 580.774,Z 766.425,A -85,B 0,C 180,E1 -1902.16,E2 -1902.16} C_VEL
LIN {X 0,Y 580.832,Z 754.056,A -85,B 0,C 180,E1 -1902.38,E2 -1902.38} C_VEL
LIN {X 0,Y 580.812,Z 654.125,A -85,B 0,C 180,E1 -1903.623,E2 -1903.623} C_VEL
LIN {X 0,Y 580.411,Z 651.401,A -85,B 0,C 180,E1 -1903.68,E2 -1903.68} C_VEL
LIN {X 0,Y 580.601,Z 628.846,A -85,B 0,C 180,E1 -1906.708,E2 -1906.708} C_VEL
LIN {X 0,Y 580.776,Z 608.483,A -85,B 0,C 180,E1 -1909.481,E2 -1909.481} C_VEL
LIN {X 0,Y 580.99,Z 587.41,A -85,B 0,C 180,E1 -1912.399,E2 -1912.399} C_VEL
LIN {X 0,Y 581.227,Z 567.361,A -85,B 0,C 180,E1 -1915.229,E2 -1915.229} C_VEL
LIN {X 0,Y 581.499,Z 547.583,A -85,B 0,C 180,E1 -1918.081,E2 -1918.081} C_VEL
LIN {X 0,Y 581.394,Z 536.681,A -85,B 0,C 180,E1 -1919.5,E2 -1919.5} C_VEL
LIN {X 0,Y 581.058,Z 531.682,A -85,B 0,C 180,E1 -1920.129,E2 -1920.129} C_VEL
LIN {X 0,Y 580.331,Z 528.198,A -85,B 0,C 180,E1 -1920.604,E2 -1920.604} C_VEL
LIN {X 0,Y 580.309,Z 528.199,A -85,B 0,C 180,E1 -1923.317,E2 -1923.317} C_VEL
LIN {X 0,Y 580.254,Z 528.201,A -85,B 0,C 180,E1 -1925.757,E2 -1925.757} C_VEL
LIN {X 0,Y 580.292,Z 528.196,A -85,B 0,C 180,E1 -1928.146,E2 -1928.146} C_VEL
LIN {X 0,Y 580.302,Z 528.205,A -85,B 0,C 180,E1 -1930.844,E2 -1930.844} C_VEL
LIN {X 0,Y 580.276,Z 528.198,A -85,B 0,C 180,E1 -1933.658,E2 -1933.658} C_VEL
LIN {X 0,Y 580.282,Z 528.205,A -85,B 0,C 180,E1 -1936.609,E2 -1936.609} C_VEL
LIN {X 0,Y 580.303,Z 528.198,A -85,B 0,C 180,E1 -1939.157,E2 -1939.157} C_VEL
LIN {X 0,Y 580.295,Z 528.196,A -85,B 0,C 180,E1 -1941.927,E2 -1941.927} C_VEL
LIN {X 0,Y 580.255,Z 528.208,A -85,B 0,C 180,E1 -1944.453,E2 -1944.453} C_VEL
LIN {X 0,Y 580.295,Z 528.2,A -85,B 0,C 180,E1 -1946.975,E2 -1946.975} C_VEL
LIN {X 0,Y 580.307,Z 528.194,A -85,B 0,C 180,E1 -1949.425,E2 -1949.425} C_VEL
LIN {X 0,Y 580.301,Z 528.199,A -85,B 0,C 180,E1 -1952.141,E2 -1952.141} C_VEL
LIN {X 0,Y 580.326,Z 528.193,A -85,B 0,C 180,E1 -1955.27,E2 -1955.27} C_VEL
LIN {X 0,Y 580.27,Z 528.202,A -85,B 0,C 180,E1 -1957.947,E2 -1957.947} C_VEL
LIN {X 0,Y 580.304,Z 528.198,A -85,B 0,C 180,E1 -1960.913,E2 -1960.913} C_VEL
LIN {X 0,Y 580.277,Z 528.202,A -85,B 0,C 180,E1 -1963.825,E2 -1963.825} C_VEL
LIN {X 0,Y 580.289,Z 528.232,A -85,B 0,C 180,E1 -1965.266,E2 -1965.266} C_VEL
LIN {X 0,Y 581.597,Z 532.481,A -85,B 0,C 180,E1 -1965.361,E2 -1965.361} C_VEL
LIN {X 0,Y 581.48,Z 568.683,A -85,B 0,C 180,E1 -1965.841,E2 -1965.841} C_VEL
LIN {X 0,Y 581.417,Z 583.595,A -85,B 0,C 180,E1 -1966.166,E2 -1966.166} C_VEL
LIN {X 0,Y 581.258,Z 599.471,A -85,B 0,C 180,E1 -1966.674,E2 -1966.674} C_VEL
LIN {X 0,Y 581.117,Z 613.125,A -85,B 0,C 180,E1 -1967.249,E2 -1967.249} C_VEL
LIN {X 0,Y 580.958,Z 626.513,A -85,B 0,C 180,E1 -1967.955,E2 -1967.955} C_VEL
LIN {X 0,Y 580.797,Z 640.097,A -85,B 0,C 180,E1 -1968.836,E2 -1968.836} C_VEL
LIN {X 0,Y 580.632,Z 652.456,A -85,B 0,C 180,E1 -1969.803,E2 -1969.803} C_VEL
LIN {X 0,Y 580.476,Z 664.555,A -85,B 0,C 180,E1 -1970.944,E2 -1970.944} C_VEL
LIN {X 0,Y 580.331,Z 675.353,A -85,B 0,C 180,E1 -1972.169,E2 -1972.169} C_VEL
LIN {X 0,Y 580.241,Z 683.833,A -85,B 0,C 180,E1 -1973.317,E2 -1973.317} C_VEL
LIN {X 0,Y 580.154,Z 690.833,A -85,B 0,C 180,E1 -1974.438,E2 -1974.438} C_VEL
LIN {X 0,Y 580.147,Z 696.399,A -85,B 0,C 180,E1 -1975.483,E2 -1975.483} C_VEL
LIN {X 0,Y 580.115,Z 702.474,A -85,B 0,C 180,E1 -1976.875,E2 -1976.875} C_VEL
LIN {X 0,Y 580.084,Z 707.156,A -85,B 0,C 180,E1 -1978.264,E2 -1978.264} C_VEL
LIN {X 0,Y 580.042,Z 709.842,A -85,B 0,C 180,E1 -1979.305,E2 -1979.305} C_VEL
LIN {X 0,Y 580.034,Z 712.363,A -85,B 0,C 180,E1 -1980.694,E2 -1980.694} C_VEL
LIN {X 0,Y 580.033,Z 713.711,A -85,B 0,C 180,E1 -1982.083,E2 -1982.083} C_VEL
LIN {X 0,Y 580.074,Z 713.917,A -85,B 0,C 180,E1 -1983.473,E2 -1983.473} C_VEL
LIN {X 0,Y 580.026,Z 713.002,A -85,B 0,C 180,E1 -1984.865,E2 -1984.865} C_VEL
LIN {X 0,Y 580.063,Z 710.932,A -85,B 0,C 180,E1 -1986.26,E2 -1986.26} C_VEL
LIN {X 0,Y 580.08,Z 707.645,A -85,B 0,C 180,E1 -1987.658,E2 -1987.658} C_VEL
LIN {X 0,Y 580.07,Z 703.058,A -85,B 0,C 180,E1 -1989.062,E2 -1989.062} C_VEL
LIN {X 0,Y 580.119,Z 697.058,A -85,B 0,C 180,E1 -1990.47,E2 -1990.47} C_VEL
LIN {X 0,Y 580.209,Z 689.491,A -85,B 0,C 180,E1 -1991.883,E2 -1991.883} C_VEL
LIN {X 0,Y 580.257,Z 681.375,A -85,B 0,C 180,E1 -1993.126,E2 -1993.126} C_VEL
LIN {X 0,Y 580.37,Z 671.719,A -85,B 0,C 180,E1 -1994.358,E2 -1994.358} C_VEL
LIN {X 0,Y 580.494,Z 661.555,A -85,B 0,C 180,E1 -1995.447,E2 -1995.447} C_VEL
LIN {X 0,Y 580.654,Z 649.608,A -85,B 0,C 180,E1 -1996.525,E2 -1996.525} C_VEL
LIN {X 0,Y 580.77,Z 637.519,A -85,B 0,C 180,E1 -1997.437,E2 -1997.437} C_VEL
LIN {X 0,Y 580.951,Z 624.655,A -85,B 0,C 180,E1 -1998.241,E2 -1998.241} C_VEL
LIN {X 0,Y 580.964,Z 623.255,A -85,B 0,C 180,E1 -1998.32,E2 -1998.32} C_VEL
LIN {X 0,Y 580.384,Z 618.176,A -85,B 0,C 180,E1 -1998.614,E2 -1998.614} C_VEL
LIN {X 0,Y 577.731,Z 609.928,A -85,B 0,C 180,E1 -1999.093,E2 -1999.093} C_VEL
LIN {X 0,Y 575.073,Z 601.446,A -85,B 0,C 180,E1 -1999.526,E2 -1999.526} C_VEL
LIN {X 0,Y 574.477,Z 596.006,A -85,B 0,C 180,E1 -1999.745,E2 -1999.745} C_VEL
LIN {X 0,Y 574.622,Z 580.428,A -85,B 0,C 180,E1 -2000.213,E2 -2000.213} C_VEL
LIN {X 0,Y 574.774,Z 565.456,A -85,B 0,C 180,E1 -2000.511,E2 -2000.511} C_VEL
LIN {X 0,Y 574.706,Z 533.332,A -85,B 0,C 180,E1 -2000.937,E2 -2000.937} C_VEL
LIN {X 0,Y 573.273,Z 529.073,A -85,B 0,C 180,E1 -2001.054,E2 -2001.054} C_VEL
LIN {X 0,Y 573.23,Z 529.085,A -85,B 0,C 180,E1 -2003.865,E2 -2003.865} C_VEL
LIN {X 0,Y 573.237,Z 529.077,A -85,B 0,C 180,E1 -2006.492,E2 -2006.492} C_VEL
LIN {X 0,Y 573.239,Z 529.076,A -85,B 0,C 180,E1 -2008.564,E2 -2008.564} C_VEL
LIN {X 0,Y 573.227,Z 529.075,A -85,B 0,C 180,E1 -2010.993,E2 -2010.993} C_VEL
LIN {X 0,Y 573.264,Z 529.072,A -85,B 0,C 180,E1 -2013.524,E2 -2013.524} C_VEL
LIN {X 0,Y 573.215,Z 529.085,A -85,B 0,C 180,E1 -2016.051,E2 -2016.051} C_VEL
LIN {X 0,Y 573.25,Z 529.075,A -85,B 0,C 180,E1 -2018.701,E2 -2018.701} C_VEL
LIN {X 0,Y 573.244,Z 529.074,A -85,B 0,C 180,E1 -2021.594,E2 -2021.594} C_VEL
LIN {X 0,Y 573.238,Z 529.084,A -85,B 0,C 180,E1 -2024.333,E2 -2024.333} C_VEL
LIN {X 0,Y 573.24,Z 529.073,A -85,B 0,C 180,E1 -2027.358,E2 -2027.358} C_VEL
LIN {X 0,Y 573.247,Z 529.083,A -85,B 0,C 180,E1 -2030.393,E2 -2030.393} C_VEL
LIN {X 0,Y 573.252,Z 529.073,A -85,B 0,C 180,E1 -2033.077,E2 -2033.077} C_VEL
LIN {X 0,Y 573.271,Z 529.07,A -85,B 0,C 180,E1 -2035.671,E2 -2035.671} C_VEL
LIN {X 0,Y 573.249,Z 529.076,A -85,B 0,C 180,E1 -2038.185,E2 -2038.185} C_VEL
LIN {X 0,Y 573.264,Z 529.081,A -85,B 0,C 180,E1 -2040.634,E2 -2040.634} C_VEL
LIN {X 0,Y 573.251,Z 529.076,A -85,B 0,C 180,E1 -2043.024,E2 -2043.024} C_VEL
